Staubli VAL3: readText.dtx

public bool bBYPASS
public bool bCycle = true
public bool bCycleEnd
bool bGetSpeed = true
bool bReadEnd
bool bReadWait
public bool bResumeCycle
bool bTxtHeadOk
public bool bWriteEnd = true
frame fPrdFrame = {x=1612.648, y=43.392, z=-88.763, rx=0.062, ry=-0.933, rz=-75.763, fatherId=world[0]}
jointRx jJointRead[100]
  [0] = {j1=8.22, j2=20.1, j3=107.19, j4=-141.77, j5=44.38, j6=150.9}
  [1] = {j1=8.22, j2=20.1, j3=107.19, j4=-141.77, j5=44.38, j6=150.9}
  [2] = {j1=10.229, j2=35.494, j3=107.593, j4=-158.624, j5=56.663, j6=165.836}
  [3] = {j1=10.423, j2=28.404, j3=105.415, j4=-155.608, j5=48.169, j6=161.142}
  [4] = {j1=-54.223, j2=64.586, j3=41.499, j4=-84.729, j5=-54.881, j6=28.938}
  [5] = {j1=-45.629, j2=26.921, j3=105.631, j4=-78.314, j5=-77.561, j6=-12.796}
  [6] = {j3=109.005, j4=80.751, j5=91.42, j6=-238.352}
  [7] = {j3=63.424, j4=82.395, j5=93.028, j6=-198.425}
  [8] = {j3=109.358, j4=80.375, j5=92.272, j6=-239.01}
  [9] = {j3=62.177, j4=82.615, j5=93.831, j6=-197.649}
public jointRx jPrdHome = {j1=40.635, j2=24.616, j3=104.715, j4=-108.663, j5=68.526, j6=132.709}
mdesc mNomSpeed = {accel=16, vel=40, decel=16, tmax=80, blend=off, leave=20, reach=20}
public mdesc mSpdOfJnt[100]
  [0] = {accel=16, vel=40, decel=16, rmax=1000, tmax=200, blend=cartesian, leave=2, reach=2}
  [1] = {accel=16, vel=40, decel=16, rmax=1000, tmax=200, blend=cartesian, leave=2, reach=2}
  [2] = {accel=16, vel=40, decel=16, rmax=1000, tmax=200, blend=cartesian, leave=2, reach=2}
  [3] = {accel=16, vel=40, decel=16, rmax=1000, tmax=200, blend=cartesian, leave=2, reach=2}
  [4] = {accel=16, vel=40, decel=16, rmax=1000, tmax=200, blend=cartesian, leave=2, reach=2}
  [5] = {accel=16, vel=40, decel=16, rmax=1000, tmax=200, blend=cartesian, leave=2, reach=2}
  [6] = {accel=16, vel=40, decel=16, rmax=1000, tmax=200, blend=cartesian, leave=2, reach=2}
  [7] = {accel=16, vel=40, decel=16, rmax=1000, tmax=200, blend=cartesian, leave=2, reach=2}
  [8] = {accel=16, vel=40, decel=16, rmax=1000, tmax=200, blend=cartesian, leave=2, reach=2}
  [9] = {accel=16, vel=40, decel=16, rmax=1000, tmax=200, blend=cartesian, leave=2, reach=2}
  [10] = {accel=16, vel=40, decel=16, rmax=1000, tmax=200, blend=cartesian, leave=2, reach=2}
  [11] = {accel=16, vel=40, decel=16, rmax=1000, tmax=200, blend=cartesian, leave=2, reach=2}
  [12] = {accel=16, vel=40, decel=16, rmax=1000, tmax=200, blend=cartesian, leave=2, reach=2}
  [13] = {accel=16, vel=40, decel=16, rmax=1000, tmax=200, blend=cartesian, leave=2, reach=2}
  [14] = {accel=16, vel=40, decel=16, rmax=1000, tmax=200, blend=cartesian, leave=2, reach=2}
  [15] = {accel=16, vel=40, decel=16, rmax=1000, tmax=200, blend=cartesian, leave=2, reach=2}
  [16] = {accel=16, vel=40, decel=16, rmax=1000, tmax=200, blend=cartesian, leave=2, reach=2}
  [17] = {accel=16, vel=40, decel=16, rmax=1000, tmax=200, blend=cartesian, leave=2, reach=2}
  [18] = {accel=16, vel=40, decel=16, rmax=1000, tmax=200, blend=cartesian, leave=2, reach=2}
  [19] = {accel=16, vel=40, decel=16, rmax=1000, tmax=200, blend=cartesian, leave=2, reach=2}
  [20] = {accel=16, vel=40, decel=16, rmax=1000, tmax=200, blend=cartesian, leave=2, reach=2}
  [21] = {accel=16, vel=40, decel=16, rmax=1000, tmax=200, blend=cartesian, leave=2, reach=2}
  [22] = {accel=16, vel=40, decel=16, rmax=1000, tmax=200, blend=cartesian, leave=2, reach=2}
  [23] = {accel=16, vel=40, decel=16, rmax=1000, tmax=200, blend=cartesian, leave=2, reach=2}
  [24] = {accel=16, vel=40, decel=16, rmax=1000, tmax=200, blend=cartesian, leave=2, reach=2}
  [25] = {accel=16, vel=40, decel=16, rmax=1000, tmax=200, blend=cartesian, leave=2, reach=2}
  [26] = {accel=16, vel=40, decel=16, rmax=1000, tmax=200, blend=cartesian, leave=2, reach=2}
  [27] = {accel=16, vel=40, decel=16, rmax=1000, tmax=200, blend=cartesian, leave=2, reach=2}
  [28] = {accel=16, vel=40, decel=16, rmax=1000, tmax=200, blend=cartesian, leave=2, reach=2}
  [29] = {accel=16, vel=40, decel=16, rmax=1000, tmax=200, blend=cartesian, leave=2, reach=2}
  [30] = {accel=16, vel=40, decel=16, rmax=1000, tmax=200, blend=cartesian, leave=2, reach=2}
  [31] = {accel=16, vel=40, decel=16, rmax=1000, tmax=200, blend=cartesian, leave=2, reach=2}
  [32] = {accel=16, vel=40, decel=16, rmax=1000, tmax=200, blend=cartesian, leave=2, reach=2}
  [33] = {accel=16, vel=40, decel=16, rmax=1000, tmax=200, blend=cartesian, leave=2, reach=2}
  [34] = {accel=16, vel=40, decel=16, rmax=1000, tmax=200, blend=cartesian, leave=2, reach=2}
  [35] = {accel=16, vel=40, decel=16, rmax=1000, tmax=200, blend=cartesian, leave=2, reach=2}
  [36] = {accel=16, vel=40, decel=16, rmax=1000, tmax=200, blend=cartesian, leave=2, reach=2}
  [37] = {accel=16, vel=40, decel=16, rmax=1000, tmax=200, blend=cartesian, leave=2, reach=2}
  [38] = {accel=16, vel=40, decel=16, rmax=1000, tmax=200, blend=cartesian, leave=2, reach=2}
  [39] = {accel=16, vel=40, decel=16, rmax=1000, tmax=200, blend=cartesian, leave=2, reach=2}
  [40] = {accel=16, vel=40, decel=16, rmax=1000, tmax=200, blend=cartesian, leave=2, reach=2}
  [41] = {accel=16, vel=40, decel=16, rmax=1000, tmax=200, blend=cartesian, leave=2, reach=2}
  [42] = {accel=16, vel=40, decel=16, rmax=1000, tmax=200, blend=cartesian, leave=2, reach=2}
  [43] = {accel=16, vel=40, decel=16, rmax=1000, tmax=200, blend=cartesian, leave=2, reach=2}
  [44] = {accel=16, vel=40, decel=16, rmax=1000, tmax=200, blend=cartesian, leave=2, reach=2}
  [45] = {accel=16, vel=40, decel=16, rmax=1000, tmax=200, blend=cartesian, leave=2, reach=2}
  [46] = {accel=16, vel=40, decel=16, rmax=1000, tmax=200, blend=cartesian, leave=2, reach=2}
  [47] = {accel=16, vel=40, decel=16, rmax=1000, tmax=200, blend=cartesian, leave=2, reach=2}
  [48] = {accel=16, vel=40, decel=16, rmax=1000, tmax=200, blend=cartesian, leave=2, reach=2}
  [49] = {accel=16, vel=40, decel=16, rmax=1000, tmax=200, blend=cartesian, leave=2, reach=2}
  [50] = {accel=16, vel=40, decel=16, rmax=1000, tmax=200, blend=cartesian, leave=2, reach=2}
  [51] = {accel=16, vel=40, decel=16, rmax=1000, tmax=200, blend=cartesian, leave=2, reach=2}
  [52] = {accel=16, vel=40, decel=16, rmax=1000, tmax=200, blend=cartesian, leave=2, reach=2}
  [53] = {accel=16, vel=40, decel=16, rmax=1000, tmax=200, blend=cartesian, leave=2, reach=2}
  [54] = {accel=16, vel=40, decel=16, rmax=1000, tmax=200, blend=cartesian, leave=2, reach=2}
  [55] = {accel=16, vel=40, decel=16, rmax=1000, tmax=200, blend=cartesian, leave=2, reach=2}
  [56] = {accel=16, vel=40, decel=16, rmax=1000, tmax=200, blend=cartesian, leave=2, reach=2}
  [57] = {accel=16, vel=40, decel=16, rmax=1000, tmax=200, blend=cartesian, leave=2, reach=2}
  [58] = {accel=16, vel=40, decel=16, rmax=1000, tmax=200, blend=cartesian, leave=2, reach=2}
  [59] = {accel=16, vel=40, decel=16, rmax=1000, tmax=200, blend=cartesian, leave=2, reach=2}
  [60] = {accel=16, vel=40, decel=16, rmax=1000, tmax=200, blend=cartesian, leave=2, reach=2}
  [61] = {accel=16, vel=40, decel=16, rmax=1000, tmax=200, blend=cartesian, leave=2, reach=2}
  [62] = {accel=16, vel=40, decel=16, rmax=1000, tmax=200, blend=cartesian, leave=2, reach=2}
  [63] = {accel=16, vel=40, decel=16, rmax=1000, tmax=200, blend=cartesian, leave=2, reach=2}
  [64] = {accel=16, vel=40, decel=16, rmax=1000, tmax=200, blend=cartesian, leave=2, reach=2}
  [65] = {accel=16, vel=40, decel=16, rmax=1000, tmax=200, blend=cartesian, leave=2, reach=2}
  [66] = {accel=16, vel=40, decel=16, rmax=1000, tmax=200, blend=cartesian, leave=2, reach=2}
  [67] = {accel=16, vel=40, decel=16, rmax=1000, tmax=200, blend=cartesian, leave=2, reach=2}
  [68] = {accel=16, vel=40, decel=16, rmax=1000, tmax=200, blend=cartesian, leave=2, reach=2}
  [69] = {accel=16, vel=40, decel=16, rmax=1000, tmax=200, blend=cartesian, leave=2, reach=2}
  [70] = {accel=16, vel=40, decel=16, rmax=1000, tmax=200, blend=cartesian, leave=2, reach=2}
  [71] = {accel=16, vel=40, decel=16, rmax=1000, tmax=200, blend=cartesian, leave=2, reach=2}
  [72] = {accel=16, vel=40, decel=16, rmax=1000, tmax=200, blend=cartesian, leave=2, reach=2}
  [73] = {accel=16, vel=40, decel=16, rmax=1000, tmax=200, blend=cartesian, leave=2, reach=2}
  [74] = {accel=16, vel=40, decel=16, rmax=1000, tmax=200, blend=cartesian, leave=2, reach=2}
  [75] = {accel=16, vel=40, decel=16, rmax=1000, tmax=200, blend=cartesian, leave=2, reach=2}
  [76] = {accel=16, vel=40, decel=16, rmax=1000, tmax=200, blend=cartesian, leave=2, reach=2}
  [77] = {accel=16, vel=40, decel=16, rmax=1000, tmax=200, blend=cartesian, leave=2, reach=2}
  [78] = {accel=16, vel=40, decel=16, rmax=1000, tmax=200, blend=cartesian, leave=2, reach=2}
  [79] = {accel=16, vel=40, decel=16, rmax=1000, tmax=200, blend=cartesian, leave=2, reach=2}
  [80] = {accel=16, vel=40, decel=16, rmax=1000, tmax=200, blend=cartesian, leave=2, reach=2}
  [81] = {accel=16, vel=40, decel=16, rmax=1000, tmax=200, blend=cartesian, leave=2, reach=2}
  [82] = {accel=16, vel=40, decel=16, rmax=1000, tmax=200, blend=cartesian, leave=2, reach=2}
  [83] = {accel=16, vel=40, decel=16, rmax=1000, tmax=200, blend=cartesian, leave=2, reach=2}
  [84] = {accel=16, vel=40, decel=16, rmax=1000, tmax=200, blend=cartesian, leave=2, reach=2}
  [85] = {accel=16, vel=40, decel=16, rmax=1000, tmax=200, blend=cartesian, leave=2, reach=2}
  [86] = {accel=16, vel=40, decel=16, rmax=1000, tmax=200, blend=cartesian, leave=2, reach=2}
  [87] = {accel=16, vel=40, decel=16, rmax=1000, tmax=200, blend=cartesian, leave=2, reach=2}
  [88] = {accel=16, vel=40, decel=16, rmax=1000, tmax=200, blend=cartesian, leave=2, reach=2}
  [89] = {accel=16, vel=40, decel=16, rmax=1000, tmax=200, blend=cartesian, leave=2, reach=2}
  [90] = {accel=16, vel=40, decel=16, rmax=1000, tmax=200, blend=cartesian, leave=2, reach=2}
  [91] = {accel=16, vel=40, decel=16, rmax=1000, tmax=200, blend=cartesian, leave=2, reach=2}
  [92] = {accel=16, vel=40, decel=16, rmax=1000, tmax=200, blend=cartesian, leave=2, reach=2}
  [93] = {accel=16, vel=40, decel=16, rmax=1000, tmax=200, blend=cartesian, leave=2, reach=2}
  [94] = {accel=16, vel=40, decel=16, rmax=1000, tmax=200, blend=cartesian, leave=2, reach=2}
  [95] = {accel=16, vel=40, decel=16, rmax=1000, tmax=200, blend=cartesian, leave=2, reach=2}
  [96] = {accel=16, vel=40, decel=16, rmax=1000, tmax=200, blend=cartesian, leave=2, reach=2}
  [97] = {accel=16, vel=40, decel=16, rmax=1000, tmax=200, blend=cartesian, leave=2, reach=2}
  [98] = {accel=16, vel=40, decel=16, rmax=1000, tmax=200, blend=cartesian, leave=2, reach=2}
  [99] = {accel=16, vel=40, decel=16, rmax=1000, tmax=200, blend=cartesian, leave=2, reach=2}
public mdesc mSpdOfPt[1000]
  [0] = {accel=40, decel=4000, tmax=15.672, leave=0, reach=0.5}
  [1] = {accel=40, decel=4000, tmax=16.369, leave=0, reach=0.5}
  [2] = {accel=40, decel=4000, tmax=17.023, leave=0, reach=0.5}
  [3] = {accel=40, decel=4000, tmax=17.611, leave=0, reach=0.5}
  [4] = {accel=40, decel=4000, tmax=18.123, leave=0, reach=0.5}
  [5] = {accel=40, decel=4000, tmax=18.562, leave=0, reach=0.5}
  [6] = {accel=40, decel=4000, tmax=18.942, leave=0, reach=0.5}
  [7] = {accel=40, decel=4000, tmax=19.269, leave=0, reach=0.5}
  [8] = {accel=40, decel=4000, tmax=19.551, leave=0, reach=0.5}
  [9] = {accel=40, decel=4000, tmax=19.789, leave=0, reach=0.5}
  [10] = {accel=40, decel=4000, tmax=19.988, leave=0, reach=0.5}
  [11] = {accel=40, decel=4000, tmax=20.148, leave=0, reach=0.5}
  [12] = {accel=40, decel=4000, tmax=20.275, leave=0, reach=0.5}
  [13] = {accel=40, decel=4000, tmax=20.376, leave=0, reach=0.5}
  [14] = {accel=40, decel=4000, tmax=20.455, leave=0, reach=0.5}
  [15] = {accel=40, decel=4000, tmax=20.517, leave=0, reach=0.5}
  [16] = {accel=40, decel=4000, tmax=20.563, leave=0, reach=0.5}
  [17] = {accel=40, decel=4000, tmax=20.596, leave=0, reach=0.5}
  [18] = {accel=40, decel=4000, tmax=20.615, leave=0, reach=0.5}
  [19] = {accel=40, decel=4000, tmax=20.621, leave=0, reach=0.5}
  [20] = {accel=40, decel=4000, tmax=20.615, leave=0, reach=0.5}
  [21] = {accel=40, decel=4000, tmax=20.6, leave=0, reach=0.5}
  [22] = {accel=40, decel=4000, tmax=20.583, leave=0, reach=0.5}
  [23] = {accel=40, decel=4000, tmax=20.564, leave=0, reach=0.5}
  [24] = {accel=40, decel=4000, tmax=20.543, leave=0, reach=0.5}
  [25] = {accel=40, decel=4000, tmax=20.52, leave=0, reach=0.5}
  [26] = {accel=40, decel=4000, tmax=20.501, leave=0, reach=0.5}
  [27] = {accel=40, decel=4000, tmax=20.495, leave=0, reach=0.5}
  [28] = {accel=40, decel=4000, tmax=20.506, leave=0, reach=0.5}
  [29] = {accel=40, decel=4000, tmax=20.53, leave=0, reach=0.5}
  [30] = {accel=40, decel=4000, tmax=20.554, leave=0, reach=0.5}
  [31] = {accel=40, decel=4000, tmax=20.568, leave=0, reach=0.5}
  [32] = {accel=40, decel=4000, tmax=20.569, leave=0, reach=0.5}
  [33] = {accel=40, decel=4000, tmax=20.562, leave=0, reach=0.5}
  [34] = {accel=40, decel=4000, tmax=20.56, leave=0, reach=0.5}
  [35] = {accel=40, decel=4000, tmax=20.571, leave=0, reach=0.5}
  [36] = {accel=40, decel=4000, tmax=20.59, leave=0, reach=0.5}
  [37] = {accel=40, decel=4000, tmax=20.611, leave=0, reach=0.5}
  [38] = {accel=40, decel=4000, tmax=20.641, leave=0, reach=0.5}
  [39] = {accel=40, decel=4000, tmax=20.701, leave=0, reach=0.5}
  [40] = {accel=40, decel=4000, tmax=20.817, leave=0, reach=0.5}
  [41] = {accel=40, decel=4000, tmax=20.998, leave=0, reach=0.5}
  [42] = {accel=40, decel=4000, tmax=21.232, leave=0, reach=0.5}
  [43] = {accel=40, decel=4000, tmax=21.485, leave=0, reach=0.5}
  [44] = {accel=40, decel=4000, tmax=21.717, leave=0, reach=0.5}
  [45] = {accel=40, decel=4000, tmax=21.897, leave=0, reach=0.5}
  [46] = {accel=40, decel=4000, tmax=22.019, leave=0, reach=0.5}
  [47] = {accel=40, decel=4000, tmax=22.098, leave=0, reach=0.5}
  [48] = {accel=40, decel=4000, tmax=22.154, leave=0, reach=0.5}
  [49] = {accel=40, decel=4000, tmax=22.195, leave=0, reach=0.5}
  [50] = {accel=40, decel=4000, tmax=22.217, leave=0, reach=0.5}
  [51] = {accel=40, decel=4000, tmax=22.213, leave=0, reach=0.5}
  [52] = {accel=40, decel=4000, tmax=22.189, leave=0, reach=0.5}
  [53] = {accel=40, decel=4000, tmax=22.153, leave=0, reach=0.5}
  [54] = {accel=40, decel=4000, tmax=22.116, leave=0, reach=0.5}
  [55] = {accel=40, decel=4000, tmax=22.079, leave=0, reach=0.5}
  [56] = {accel=40, decel=4000, tmax=22.04, leave=0, reach=0.5}
  [57] = {accel=40, decel=4000, tmax=21.995, leave=0, reach=0.5}
  [58] = {accel=40, decel=4000, tmax=21.94, leave=0, reach=0.5}
  [59] = {accel=40, decel=4000, tmax=21.876, leave=0, reach=0.5}
  [60] = {accel=40, decel=4000, tmax=21.809, leave=0, reach=0.5}
  [61] = {accel=40, decel=4000, tmax=21.74, leave=0, reach=0.5}
  [62] = {accel=40, decel=4000, tmax=21.667, leave=0, reach=0.5}
  [63] = {accel=40, decel=4000, tmax=21.585, leave=0, reach=0.5}
  [64] = {accel=40, decel=4000, tmax=21.491, leave=0, reach=0.5}
  [65] = {accel=40, decel=4000, tmax=21.382, leave=0, reach=0.5}
  [66] = {accel=40, decel=4000, tmax=21.258, leave=0, reach=0.5}
  [67] = {accel=40, decel=4000, tmax=21.117, leave=0, reach=0.5}
  [68] = {accel=40, decel=4000, tmax=20.955, leave=0, reach=0.5}
  [69] = {accel=40, decel=4000, tmax=20.766, leave=0, reach=0.5}
  [70] = {accel=40, decel=4000, tmax=20.55, leave=0, reach=0.5}
  [71] = {accel=40, decel=4000, tmax=20.313, leave=0, reach=0.5}
  [72] = {accel=40, decel=4000, tmax=20.06, leave=0, reach=0.5}
  [73] = {accel=40, decel=4000, tmax=19.795, leave=0, reach=0.5}
  [74] = {accel=40, decel=4000, tmax=19.518, leave=0, reach=0.5}
  [75] = {accel=40, decel=4000, tmax=19.229, leave=0, reach=0.5}
  [76] = {accel=40, decel=4000, tmax=18.929, leave=0, reach=0.5}
  [77] = {accel=40, decel=4000, tmax=18.616, leave=0, reach=0.5}
  [78] = {accel=40, decel=4000, tmax=18.288, leave=0, reach=0.5}
  [79] = {accel=40, decel=4000, tmax=17.947, leave=0, reach=0.5}
  [80] = {accel=40, decel=4000, tmax=17.601, leave=0, reach=0.5}
  [81] = {accel=40, decel=4000, tmax=17.259, leave=0, reach=0.5}
  [82] = {accel=40, decel=4000, tmax=16.931, leave=0, reach=0.5}
  [83] = {accel=40, decel=4000, tmax=16.613, leave=0, reach=0.5}
  [84] = {accel=40, decel=4000, tmax=16.293, leave=0, reach=0.5}
  [85] = {accel=40, decel=4000, tmax=15.957, leave=0, reach=0.5}
  [86] = {accel=40, decel=4000, tmax=15.595, leave=0, reach=0.5}
  [87] = {accel=40, decel=4000, tmax=15.202, leave=0, reach=0.5}
  [88] = {accel=40, decel=4000, tmax=14.779, leave=0, reach=0.5}
  [89] = {accel=40, decel=4000, tmax=14.331, leave=0, reach=0.5}
  [90] = {accel=40, decel=4000, tmax=13.865, leave=0, reach=0.5}
  [91] = {accel=40, decel=4000, tmax=13.393, leave=0, reach=0.5}
  [92] = {accel=40, decel=4000, tmax=12.925, leave=0, reach=0.5}
  [93] = {accel=40, decel=4000, tmax=28.624, leave=0, reach=0.5}
  [94] = {accel=40, decel=4000, tmax=13.153, leave=0, reach=0.5}
  [95] = {accel=40, decel=4000, tmax=13.601, leave=0, reach=0.5}
  [96] = {accel=40, decel=4000, tmax=14.047, leave=0, reach=0.5}
  [97] = {accel=40, decel=4000, tmax=14.484, leave=0, reach=0.5}
  [98] = {accel=40, decel=4000, tmax=14.903, leave=0, reach=0.5}
  [99] = {accel=40, decel=4000, tmax=15.299, leave=0, reach=0.5}
  [100] = {accel=40, decel=4000, tmax=15.67, leave=0, reach=0.5}
  [101] = {accel=40, decel=4000, tmax=16.022, leave=0, reach=0.5}
  [102] = {accel=40, decel=4000, tmax=16.368, leave=0, reach=0.5}
  [103] = {accel=40, decel=4000, tmax=16.723, leave=0, reach=0.5}
  [104] = {accel=40, decel=4000, tmax=17.091, leave=0, reach=0.5}
  [105] = {accel=40, decel=4000, tmax=17.467, leave=0, reach=0.5}
  [106] = {accel=40, decel=4000, tmax=17.843, leave=0, reach=0.5}
  [107] = {accel=40, decel=4000, tmax=18.211, leave=0, reach=0.5}
  [108] = {accel=40, decel=4000, tmax=18.567, leave=0, reach=0.5}
  [109] = {accel=40, decel=4000, tmax=18.911, leave=0, reach=0.5}
  [110] = {accel=40, decel=4000, tmax=19.238, leave=0, reach=0.5}
  [111] = {accel=40, decel=4000, tmax=19.547, leave=0, reach=0.5}
  [112] = {accel=40, decel=4000, tmax=19.837, leave=0, reach=0.5}
  [113] = {accel=40, decel=4000, tmax=20.111, leave=0, reach=0.5}
  [114] = {accel=40, decel=4000, tmax=20.367, leave=0, reach=0.5}
  [115] = {accel=40, decel=4000, tmax=20.602, leave=0, reach=0.5}
  [116] = {accel=40, decel=4000, tmax=20.813, leave=0, reach=0.5}
  [117] = {accel=40, decel=4000, tmax=21.001, leave=0, reach=0.5}
  [118] = {accel=40, decel=4000, tmax=21.172, leave=0, reach=0.5}
  [119] = {accel=40, decel=4000, tmax=21.328, leave=0, reach=0.5}
  [120] = {accel=40, decel=4000, tmax=21.469, leave=0, reach=0.5}
  [121] = {accel=40, decel=4000, tmax=21.595, leave=0, reach=0.5}
  [122] = {accel=40, decel=4000, tmax=21.708, leave=0, reach=0.5}
  [123] = {accel=40, decel=4000, tmax=21.81, leave=0, reach=0.5}
  [124] = {accel=40, decel=4000, tmax=21.907, leave=0, reach=0.5}
  [125] = {accel=40, decel=4000, tmax=21.998, leave=0, reach=0.5}
  [126] = {accel=40, decel=4000, tmax=22.082, leave=0, reach=0.5}
  [127] = {accel=40, decel=4000, tmax=22.155, leave=0, reach=0.5}
  [128] = {accel=40, decel=4000, tmax=22.217, leave=0, reach=0.5}
  [129] = {accel=40, decel=4000, tmax=22.272, leave=0, reach=0.5}
  [130] = {accel=40, decel=4000, tmax=22.324, leave=0, reach=0.5}
  [131] = {accel=40, decel=4000, tmax=22.375, leave=0, reach=0.5}
  [132] = {accel=40, decel=4000, tmax=22.423, leave=0, reach=0.5}
  [133] = {accel=40, decel=4000, tmax=22.459, leave=0, reach=0.5}
  [134] = {accel=40, decel=4000, tmax=22.473, leave=0, reach=0.5}
  [135] = {accel=40, decel=4000, tmax=22.461, leave=0, reach=0.5}
  [136] = {accel=40, decel=4000, tmax=22.43, leave=0, reach=0.5}
  [137] = {accel=40, decel=4000, tmax=22.386, leave=0, reach=0.5}
  [138] = {accel=40, decel=4000, tmax=22.324, leave=0, reach=0.5}
  [139] = {accel=40, decel=4000, tmax=22.223, leave=0, reach=0.5}
  [140] = {accel=40, decel=4000, tmax=22.065, leave=0, reach=0.5}
  [141] = {accel=40, decel=4000, tmax=21.849, leave=0, reach=0.5}
  [142] = {accel=40, decel=4000, tmax=21.606, leave=0, reach=0.5}
  [143] = {accel=40, decel=4000, tmax=21.378, leave=0, reach=0.5}
  [144] = {accel=40, decel=4000, tmax=21.204, leave=0, reach=0.5}
  [145] = {accel=40, decel=4000, tmax=21.097, leave=0, reach=0.5}
  [146] = {accel=40, decel=4000, tmax=21.048, leave=0, reach=0.5}
  [147] = {accel=40, decel=4000, tmax=21.033, leave=0, reach=0.5}
  [148] = {accel=40, decel=4000, tmax=21.031, leave=0, reach=0.5}
  [149] = {accel=40, decel=4000, tmax=21.033, leave=0, reach=0.5}
  [150] = {accel=40, decel=4000, tmax=21.04, leave=0, reach=0.5}
  [151] = {accel=40, decel=4000, tmax=21.05, leave=0, reach=0.5}
  [152] = {accel=40, decel=4000, tmax=21.061, leave=0, reach=0.5}
  [153] = {accel=40, decel=4000, tmax=21.064, leave=0, reach=0.5}
  [154] = {accel=40, decel=4000, tmax=21.054, leave=0, reach=0.5}
  [155] = {accel=40, decel=4000, tmax=21.033, leave=0, reach=0.5}
  [156] = {accel=40, decel=4000, tmax=21.011, leave=0, reach=0.5}
  [157] = {accel=40, decel=4000, tmax=20.997, leave=0, reach=0.5}
  [158] = {accel=40, decel=4000, tmax=20.992, leave=0, reach=0.5}
  [159] = {accel=40, decel=4000, tmax=20.987, leave=0, reach=0.5}
  [160] = {accel=40, decel=4000, tmax=20.974, leave=0, reach=0.5}
  [161] = {accel=40, decel=4000, tmax=20.952, leave=0, reach=0.5}
  [162] = {accel=40, decel=4000, tmax=20.927, leave=0, reach=0.5}
  [163] = {accel=40, decel=4000, tmax=20.9, leave=0, reach=0.5}
  [164] = {accel=40, decel=4000, tmax=20.867, leave=0, reach=0.5}
  [165] = {accel=40, decel=4000, tmax=20.817, leave=0, reach=0.5}
  [166] = {accel=40, decel=4000, tmax=20.744, leave=0, reach=0.5}
  [167] = {accel=40, decel=4000, tmax=20.65, leave=0, reach=0.5}
  [168] = {accel=40, decel=4000, tmax=20.537, leave=0, reach=0.5}
  [169] = {accel=40, decel=4000, tmax=20.405, leave=0, reach=0.5}
  [170] = {accel=40, decel=4000, tmax=20.254, leave=0, reach=0.5}
  [171] = {accel=40, decel=4000, tmax=20.081, leave=0, reach=0.5}
  [172] = {accel=40, decel=4000, tmax=19.882, leave=0, reach=0.5}
  [173] = {accel=40, decel=4000, tmax=19.655, leave=0, reach=0.5}
  [174] = {accel=40, decel=4000, tmax=19.393, leave=0, reach=0.5}
  [175] = {accel=40, decel=4000, tmax=19.098, leave=0, reach=0.5}
  [176] = {accel=40, decel=4000, tmax=18.769, leave=0, reach=0.5}
  [177] = {accel=40, decel=4000, tmax=18.404, leave=0, reach=0.5}
  [178] = {accel=40, decel=4000, tmax=17.999, leave=0, reach=0.5}
  [179] = {accel=40, decel=4000, tmax=17.549, leave=0, reach=0.5}
  [180] = {accel=40, decel=4000, tmax=17.05, leave=0, reach=0.5}
  [181] = {accel=40, decel=4000, tmax=16.497, leave=0, reach=0.5}
  [182] = {accel=40, decel=4000, tmax=15.886, leave=0, reach=0.5}
  [183] = {accel=40, decel=4000, tmax=34.921, leave=0, reach=0.5}
  [184] = {accel=40, decel=4000, tmax=15.966, leave=0, reach=0.5}
  [185] = {accel=40, decel=4000, tmax=16.507, leave=0, reach=0.5}
  [186] = {accel=40, decel=4000, tmax=17.012, leave=0, reach=0.5}
  [187] = {accel=40, decel=4000, tmax=17.481, leave=0, reach=0.5}
  [188] = {accel=40, decel=4000, tmax=17.915, leave=0, reach=0.5}
  [189] = {accel=40, decel=4000, tmax=18.317, leave=0, reach=0.5}
  [190] = {accel=40, decel=4000, tmax=18.687, leave=0, reach=0.5}
  [191] = {accel=40, decel=4000, tmax=19.026, leave=0, reach=0.5}
  [192] = {accel=40, decel=4000, tmax=19.333, leave=0, reach=0.5}
  [193] = {accel=40, decel=4000, tmax=19.612, leave=0, reach=0.5}
  [194] = {accel=40, decel=4000, tmax=19.868, leave=0, reach=0.5}
  [195] = {accel=40, decel=4000, tmax=20.105, leave=0, reach=0.5}
  [196] = {accel=40, decel=4000, tmax=20.322, leave=0, reach=0.5}
  [197] = {accel=40, decel=4000, tmax=20.52, leave=0, reach=0.5}
  [198] = {accel=40, decel=4000, tmax=20.694, leave=0, reach=0.5}
  [199] = {accel=40, decel=4000, tmax=20.835, leave=0, reach=0.5}
  [200] = {accel=40, decel=4000, tmax=20.941, leave=0, reach=0.5}
  [201] = {accel=40, decel=4000, tmax=21.018, leave=0, reach=0.5}
  [202] = {accel=40, decel=4000, tmax=21.084, leave=0, reach=0.5}
  [203] = {accel=40, decel=4000, tmax=21.153, leave=0, reach=0.5}
  [204] = {accel=40, decel=4000, tmax=21.221, leave=0, reach=0.5}
  [205] = {accel=40, decel=4000, tmax=21.279, leave=0, reach=0.5}
  [206] = {accel=40, decel=4000, tmax=21.32, leave=0, reach=0.5}
  [207] = {accel=40, decel=4000, tmax=21.347, leave=0, reach=0.5}
  [208] = {accel=40, decel=4000, tmax=21.367, leave=0, reach=0.5}
  [209] = {accel=40, decel=4000, tmax=21.386, leave=0, reach=0.5}
  [210] = {accel=40, decel=4000, tmax=21.4, leave=0, reach=0.5}
  [211] = {accel=40, decel=4000, tmax=21.406, leave=0, reach=0.5}
  [212] = {accel=40, decel=4000, tmax=21.403, leave=0, reach=0.5}
  [213] = {accel=40, decel=4000, tmax=21.393, leave=0, reach=0.5}
  [214] = {accel=40, decel=4000, tmax=21.381, leave=0, reach=0.5}
  [215] = {accel=40, decel=4000, tmax=21.369, leave=0, reach=0.5}
  [216] = {accel=40, decel=4000, tmax=21.359, leave=0, reach=0.5}
  [217] = {accel=40, decel=4000, tmax=21.354, leave=0, reach=0.5}
  [218] = {accel=40, decel=4000, tmax=21.364, leave=0, reach=0.5}
  [219] = {accel=40, decel=4000, tmax=21.408, leave=0, reach=0.5}
  [220] = {accel=40, decel=4000, tmax=21.506, leave=0, reach=0.5}
  [221] = {accel=40, decel=4000, tmax=21.663, leave=0, reach=0.5}
  [222] = {accel=40, decel=4000, tmax=21.866, leave=0, reach=0.5}
  [223] = {accel=40, decel=4000, tmax=22.075, leave=0, reach=0.5}
  [224] = {accel=40, decel=4000, tmax=22.25, leave=0, reach=0.5}
  [225] = {accel=40, decel=4000, tmax=22.368, leave=0, reach=0.5}
  [226] = {accel=40, decel=4000, tmax=22.439, leave=0, reach=0.5}
  [227] = {accel=40, decel=4000, tmax=22.485, leave=0, reach=0.5}
  [228] = {accel=40, decel=4000, tmax=22.523, leave=0, reach=0.5}
  [229] = {accel=40, decel=4000, tmax=22.553, leave=0, reach=0.5}
  [230] = {accel=40, decel=4000, tmax=22.566, leave=0, reach=0.5}
  [231] = {accel=40, decel=4000, tmax=22.552, leave=0, reach=0.5}
  [232] = {accel=40, decel=4000, tmax=22.512, leave=0, reach=0.5}
  [233] = {accel=40, decel=4000, tmax=22.455, leave=0, reach=0.5}
  [234] = {accel=40, decel=4000, tmax=22.392, leave=0, reach=0.5}
  [235] = {accel=40, decel=4000, tmax=22.327, leave=0, reach=0.5}
  [236] = {accel=40, decel=4000, tmax=22.257, leave=0, reach=0.5}
  [237] = {accel=40, decel=4000, tmax=22.178, leave=0, reach=0.5}
  [238] = {accel=40, decel=4000, tmax=22.085, leave=0, reach=0.5}
  [239] = {accel=40, decel=4000, tmax=21.979, leave=0, reach=0.5}
  [240] = {accel=40, decel=4000, tmax=21.864, leave=0, reach=0.5}
  [241] = {accel=40, decel=4000, tmax=21.743, leave=0, reach=0.5}
  [242] = {accel=40, decel=4000, tmax=21.613, leave=0, reach=0.5}
  [243] = {accel=40, decel=4000, tmax=21.472, leave=0, reach=0.5}
  [244] = {accel=40, decel=4000, tmax=21.316, leave=0, reach=0.5}
  [245] = {accel=40, decel=4000, tmax=21.144, leave=0, reach=0.5}
  [246] = {accel=40, decel=4000, tmax=20.958, leave=0, reach=0.5}
  [247] = {accel=40, decel=4000, tmax=20.76, leave=0, reach=0.5}
  [248] = {accel=40, decel=4000, tmax=20.548, leave=0, reach=0.5}
  [249] = {accel=40, decel=4000, tmax=20.318, leave=0, reach=0.5}
  [250] = {accel=40, decel=4000, tmax=20.069, leave=0, reach=0.5}
  [251] = {accel=40, decel=4000, tmax=19.799, leave=0, reach=0.5}
  [252] = {accel=40, decel=4000, tmax=19.511, leave=0, reach=0.5}
  [253] = {accel=40, decel=4000, tmax=19.202, leave=0, reach=0.5}
  [254] = {accel=40, decel=4000, tmax=18.868, leave=0, reach=0.5}
  [255] = {accel=40, decel=4000, tmax=18.508, leave=0, reach=0.5}
  [256] = {accel=40, decel=4000, tmax=18.128, leave=0, reach=0.5}
  [257] = {accel=40, decel=4000, tmax=17.735, leave=0, reach=0.5}
  [258] = {accel=40, decel=4000, tmax=17.333, leave=0, reach=0.5}
  [259] = {accel=40, decel=4000, tmax=16.925, leave=0, reach=0.5}
  [260] = {accel=40, decel=4000, tmax=16.52, leave=0, reach=0.5}
  [261] = {accel=40, decel=4000, tmax=16.124, leave=0, reach=0.5}
  [262] = {accel=40, decel=4000, tmax=15.739, leave=0, reach=0.5}
  [263] = {accel=40, decel=4000, tmax=15.36, leave=0, reach=0.5}
  [264] = {accel=40, decel=4000, tmax=14.977, leave=0, reach=0.5}
  [265] = {accel=40, decel=4000, tmax=14.58, leave=0, reach=0.5}
  [266] = {accel=40, decel=4000, tmax=14.169, leave=0, reach=0.5}
  [267] = {accel=40, decel=4000, tmax=13.749, leave=0, reach=0.5}
  [268] = {accel=40, decel=4000, tmax=13.325, leave=0, reach=0.5}
  [269] = {accel=40, decel=4000, tmax=29.431, leave=0, reach=0.5}
  [270] = {accel=40, decel=4000, tmax=13.43, leave=0, reach=0.5}
  [271] = {accel=40, decel=4000, tmax=13.831, leave=0, reach=0.5}
  [272] = {accel=40, decel=4000, tmax=14.232, leave=0, reach=0.5}
  [273] = {accel=40, decel=4000, tmax=14.633, leave=0, reach=0.5}
  [274] = {accel=40, decel=4000, tmax=15.039, leave=0, reach=0.5}
  [275] = {accel=40, decel=4000, tmax=15.454, leave=0, reach=0.5}
  [276] = {accel=40, decel=4000, tmax=15.879, leave=0, reach=0.5}
  [277] = {accel=40, decel=4000, tmax=16.311, leave=0, reach=0.5}
  [278] = {accel=40, decel=4000, tmax=16.744, leave=0, reach=0.5}
  [279] = {accel=40, decel=4000, tmax=17.173, leave=0, reach=0.5}
  [280] = {accel=40, decel=4000, tmax=17.594, leave=0, reach=0.5}
  [281] = {accel=40, decel=4000, tmax=18.002, leave=0, reach=0.5}
  [282] = {accel=40, decel=4000, tmax=18.387, leave=0, reach=0.5}
  [283] = {accel=40, decel=4000, tmax=18.742, leave=0, reach=0.5}
  [284] = {accel=40, decel=4000, tmax=19.067, leave=0, reach=0.5}
  [285] = {accel=40, decel=4000, tmax=19.367, leave=0, reach=0.5}
  [286] = {accel=40, decel=4000, tmax=19.646, leave=0, reach=0.5}
  [287] = {accel=40, decel=4000, tmax=19.908, leave=0, reach=0.5}
  [288] = {accel=40, decel=4000, tmax=20.154, leave=0, reach=0.5}
  [289] = {accel=40, decel=4000, tmax=20.386, leave=0, reach=0.5}
  [290] = {accel=40, decel=4000, tmax=20.608, leave=0, reach=0.5}
  [291] = {accel=40, decel=4000, tmax=20.821, leave=0, reach=0.5}
  [292] = {accel=40, decel=4000, tmax=21.021, leave=0, reach=0.5}
  [293] = {accel=40, decel=4000, tmax=21.206, leave=0, reach=0.5}
  [294] = {accel=40, decel=4000, tmax=21.373, leave=0, reach=0.5}
  [295] = {accel=40, decel=4000, tmax=21.528, leave=0, reach=0.5}
  [296] = {accel=40, decel=4000, tmax=21.673, leave=0, reach=0.5}
  [297] = {accel=40, decel=4000, tmax=21.809, leave=0, reach=0.5}
  [298] = {accel=40, decel=4000, tmax=21.934, leave=0, reach=0.5}
  [299] = {accel=40, decel=4000, tmax=22.042, leave=0, reach=0.5}
  [300] = {accel=40, decel=4000, tmax=22.134, leave=0, reach=0.5}
  [301] = {accel=40, decel=4000, tmax=22.213, leave=0, reach=0.5}
  [302] = {accel=40, decel=4000, tmax=22.287, leave=0, reach=0.5}
  [303] = {accel=40, decel=4000, tmax=22.358, leave=0, reach=0.5}
  [304] = {accel=40, decel=4000, tmax=22.421, leave=0, reach=0.5}
  [305] = {accel=40, decel=4000, tmax=22.463, leave=0, reach=0.5}
  [306] = {accel=40, decel=4000, tmax=22.473, leave=0, reach=0.5}
  [307] = {accel=40, decel=4000, tmax=22.453, leave=0, reach=0.5}
  [308] = {accel=40, decel=4000, tmax=22.416, leave=0, reach=0.5}
  [309] = {accel=40, decel=4000, tmax=22.378, leave=0, reach=0.5}
  [310] = {accel=40, decel=4000, tmax=22.342, leave=0, reach=0.5}
  [311] = {accel=40, decel=4000, tmax=22.301, leave=0, reach=0.5}
  [312] = {accel=40, decel=4000, tmax=22.231, leave=0, reach=0.5}
  [313] = {accel=40, decel=4000, tmax=22.114, leave=0, reach=0.5}
  [314] = {accel=40, decel=4000, tmax=21.958, leave=0, reach=0.5}
  [315] = {accel=40, decel=4000, tmax=21.796, leave=0, reach=0.5}
  [316] = {accel=40, decel=4000, tmax=21.663, leave=0, reach=0.5}
  [317] = {accel=40, decel=4000, tmax=21.576, leave=0, reach=0.5}
  [318] = {accel=40, decel=4000, tmax=21.535, leave=0, reach=0.5}
  [319] = {accel=40, decel=4000, tmax=21.524, leave=0, reach=0.5}
  [320] = {accel=40, decel=4000, tmax=21.53, leave=0, reach=0.5}
  [321] = {accel=40, decel=4000, tmax=21.54, leave=0, reach=0.5}
  [322] = {accel=40, decel=4000, tmax=21.551, leave=0, reach=0.5}
  [323] = {accel=40, decel=4000, tmax=21.561, leave=0, reach=0.5}
  [324] = {accel=40, decel=4000, tmax=21.567, leave=0, reach=0.5}
  [325] = {accel=40, decel=4000, tmax=21.569, leave=0, reach=0.5}
  [326] = {accel=40, decel=4000, tmax=21.566, leave=0, reach=0.5}
  [327] = {accel=40, decel=4000, tmax=21.557, leave=0, reach=0.5}
  [328] = {accel=40, decel=4000, tmax=21.538, leave=0, reach=0.5}
  [329] = {accel=40, decel=4000, tmax=21.504, leave=0, reach=0.5}
  [330] = {accel=40, decel=4000, tmax=21.447, leave=0, reach=0.5}
  [331] = {accel=40, decel=4000, tmax=21.364, leave=0, reach=0.5}
  [332] = {accel=40, decel=4000, tmax=21.26, leave=0, reach=0.5}
  [333] = {accel=40, decel=4000, tmax=21.149, leave=0, reach=0.5}
  [334] = {accel=40, decel=4000, tmax=21.04, leave=0, reach=0.5}
  [335] = {accel=40, decel=4000, tmax=20.932, leave=0, reach=0.5}
  [336] = {accel=40, decel=4000, tmax=20.805, leave=0, reach=0.5}
  [337] = {accel=40, decel=4000, tmax=20.639, leave=0, reach=0.5}
  [338] = {accel=40, decel=4000, tmax=20.426, leave=0, reach=0.5}
  [339] = {accel=40, decel=4000, tmax=20.175, leave=0, reach=0.5}
  [340] = {accel=40, decel=4000, tmax=19.897, leave=0, reach=0.5}
  [341] = {accel=40, decel=4000, tmax=19.603, leave=0, reach=0.5}
  [342] = {accel=40, decel=4000, tmax=19.296, leave=0, reach=0.5}
  [343] = {accel=40, decel=4000, tmax=18.975, leave=0, reach=0.5}
  [344] = {accel=40, decel=4000, tmax=18.635, leave=0, reach=0.5}
  [345] = {accel=40, decel=4000, tmax=18.27, leave=0, reach=0.5}
  [346] = {accel=40, decel=4000, tmax=17.874, leave=0, reach=0.5}
  [347] = {accel=40, decel=4000, tmax=17.448, leave=0, reach=0.5}
  [348] = {accel=40, decel=4000, tmax=16.994, leave=0, reach=0.5}
  [349] = {accel=40, decel=4000, tmax=16.511, leave=0, reach=0.5}
  [350] = {accel=40, decel=4000, tmax=16.001, leave=0, reach=0.5}
  [351] = {accel=40, decel=4000, tmax=35.192, leave=0, reach=0.5}
  [352] = {accel=40, decel=4000, tmax=16.003, leave=0, reach=0.5}
  [353] = {accel=40, decel=4000, tmax=16.487, leave=0, reach=0.5}
  [354] = {accel=40, decel=4000, tmax=16.949, leave=0, reach=0.5}
  [355] = {accel=40, decel=4000, tmax=17.385, leave=0, reach=0.5}
  [356] = {accel=40, decel=4000, tmax=17.795, leave=0, reach=0.5}
  [357] = {accel=40, decel=4000, tmax=18.183, leave=0, reach=0.5}
  [358] = {accel=40, decel=4000, tmax=18.556, leave=0, reach=0.5}
  [359] = {accel=40, decel=4000, tmax=18.916, leave=0, reach=0.5}
  [360] = {accel=40, decel=4000, tmax=19.267, leave=0, reach=0.5}
  [361] = {accel=40, decel=4000, tmax=19.605, leave=0, reach=0.5}
  [362] = {accel=40, decel=4000, tmax=19.919, leave=0, reach=0.5}
  [363] = {accel=40, decel=4000, tmax=20.195, leave=0, reach=0.5}
  [364] = {accel=40, decel=4000, tmax=20.425, leave=0, reach=0.5}
  [365] = {accel=40, decel=4000, tmax=20.612, leave=0, reach=0.5}
  [366] = {accel=40, decel=4000, tmax=20.777, leave=0, reach=0.5}
  [367] = {accel=40, decel=4000, tmax=20.934, leave=0, reach=0.5}
  [368] = {accel=40, decel=4000, tmax=21.089, leave=0, reach=0.5}
  [369] = {accel=40, decel=4000, tmax=21.234, leave=0, reach=0.5}
  [370] = {accel=40, decel=4000, tmax=21.357, leave=0, reach=0.5}
  [371] = {accel=40, decel=4000, tmax=21.445, leave=0, reach=0.5}
  [372] = {accel=40, decel=4000, tmax=21.497, leave=0, reach=0.5}
  [373] = {accel=40, decel=4000, tmax=21.52, leave=0, reach=0.5}
  [374] = {accel=40, decel=4000, tmax=21.525, leave=0, reach=0.5}
  [375] = {accel=40, decel=4000, tmax=21.523, leave=0, reach=0.5}
  [376] = {accel=40, decel=4000, tmax=21.521, leave=0, reach=0.5}
  [377] = {accel=40, decel=4000, tmax=21.519, leave=0, reach=0.5}
  [378] = {accel=40, decel=4000, tmax=21.513, leave=0, reach=0.5}
  [379] = {accel=40, decel=4000, tmax=21.504, leave=0, reach=0.5}
  [380] = {accel=40, decel=4000, tmax=21.493, leave=0, reach=0.5}
  [381] = {accel=40, decel=4000, tmax=21.485, leave=0, reach=0.5}
  [382] = {accel=40, decel=4000, tmax=21.491, leave=0, reach=0.5}
  [383] = {accel=40, decel=4000, tmax=21.525, leave=0, reach=0.5}
  [384] = {accel=40, decel=4000, tmax=21.596, leave=0, reach=0.5}
  [385] = {accel=40, decel=4000, tmax=21.7, leave=0, reach=0.5}
  [386] = {accel=40, decel=4000, tmax=21.817, leave=0, reach=0.5}
  [387] = {accel=40, decel=4000, tmax=21.917, leave=0, reach=0.5}
  [388] = {accel=40, decel=4000, tmax=21.981, leave=0, reach=0.5}
  [389] = {accel=40, decel=4000, tmax=22.015, leave=0, reach=0.5}
  [390] = {accel=40, decel=4000, tmax=22.04, leave=0, reach=0.5}
  [391] = {accel=40, decel=4000, tmax=22.076, leave=0, reach=0.5}
  [392] = {accel=40, decel=4000, tmax=22.124, leave=0, reach=0.5}
  [393] = {accel=40, decel=4000, tmax=22.169, leave=0, reach=0.5}
  [394] = {accel=40, decel=4000, tmax=22.191, leave=0, reach=0.5}
  [395] = {accel=40, decel=4000, tmax=22.176, leave=0, reach=0.5}
  [396] = {accel=40, decel=4000, tmax=22.123, leave=0, reach=0.5}
  [397] = {accel=40, decel=4000, tmax=22.051, leave=0, reach=0.5}
  [398] = {accel=40, decel=4000, tmax=21.974, leave=0, reach=0.5}
  [399] = {accel=40, decel=4000, tmax=21.898, leave=0, reach=0.5}
  [400] = {accel=40, decel=4000, tmax=21.819, leave=0, reach=0.5}
  [401] = {accel=40, decel=4000, tmax=21.724, leave=0, reach=0.5}
  [402] = {accel=40, decel=4000, tmax=21.607, leave=0, reach=0.5}
  [403] = {accel=40, decel=4000, tmax=21.468, leave=0, reach=0.5}
  [404] = {accel=40, decel=4000, tmax=21.313, leave=0, reach=0.5}
  [405] = {accel=40, decel=4000, tmax=21.147, leave=0, reach=0.5}
  [406] = {accel=40, decel=4000, tmax=20.971, leave=0, reach=0.5}
  [407] = {accel=40, decel=4000, tmax=20.78, leave=0, reach=0.5}
  [408] = {accel=40, decel=4000, tmax=20.572, leave=0, reach=0.5}
  [409] = {accel=40, decel=4000, tmax=20.348, leave=0, reach=0.5}
  [410] = {accel=40, decel=4000, tmax=20.113, leave=0, reach=0.5}
  [411] = {accel=40, decel=4000, tmax=19.87, leave=0, reach=0.5}
  [412] = {accel=40, decel=4000, tmax=19.62, leave=0, reach=0.5}
  [413] = {accel=40, decel=4000, tmax=19.36, leave=0, reach=0.5}
  [414] = {accel=40, decel=4000, tmax=19.09, leave=0, reach=0.5}
  [415] = {accel=40, decel=4000, tmax=18.803, leave=0, reach=0.5}
  [416] = {accel=40, decel=4000, tmax=18.496, leave=0, reach=0.5}
  [417] = {accel=40, decel=4000, tmax=18.158, leave=0, reach=0.5}
  [418] = {accel=40, decel=4000, tmax=17.785, leave=0, reach=0.5}
  [419] = {accel=40, decel=4000, tmax=17.38, leave=0, reach=0.5}
  [420] = {accel=40, decel=4000, tmax=16.952, leave=0, reach=0.5}
  [421] = {accel=40, decel=4000, tmax=16.512, leave=0, reach=0.5}
  [422] = {accel=40, decel=4000, tmax=16.064, leave=0, reach=0.5}
  [423] = {accel=40, decel=4000, tmax=15.613, leave=0, reach=0.5}
  [424] = {accel=40, decel=4000, tmax=15.163, leave=0, reach=0.5}
  [425] = {accel=40, decel=4000, tmax=14.719, leave=0, reach=0.5}
  [426] = {accel=40, decel=4000, tmax=14.289, leave=0, reach=0.5}
  [427] = {accel=40, decel=4000, tmax=13.875, leave=0, reach=0.5}
  [428] = {accel=40, decel=4000, tmax=13.477, leave=0, reach=0.5}
  [429] = {accel=40, decel=4000, tmax=42.678, leave=0, reach=0.5}
  [430] = {accel=40, decel=4000, tmax=13.946, leave=0, reach=0.5}
  [431] = {accel=40, decel=4000, tmax=14.383, leave=0, reach=0.5}
  [432] = {accel=40, decel=4000, tmax=14.831, leave=0, reach=0.5}
  [433] = {accel=40, decel=4000, tmax=15.283, leave=0, reach=0.5}
  [434] = {accel=40, decel=4000, tmax=15.737, leave=0, reach=0.5}
  [435] = {accel=40, decel=4000, tmax=16.189, leave=0, reach=0.5}
  [436] = {accel=40, decel=4000, tmax=16.631, leave=0, reach=0.5}
  [437] = {accel=40, decel=4000, tmax=17.053, leave=0, reach=0.5}
  [438] = {accel=40, decel=4000, tmax=17.441, leave=0, reach=0.5}
  [439] = {accel=40, decel=4000, tmax=17.788, leave=0, reach=0.5}
  [440] = {accel=40, decel=4000, tmax=18.099, leave=0, reach=0.5}
  [441] = {accel=40, decel=4000, tmax=18.388, leave=0, reach=0.5}
  [442] = {accel=40, decel=4000, tmax=18.664, leave=0, reach=0.5}
  [443] = {accel=40, decel=4000, tmax=18.934, leave=0, reach=0.5}
  [444] = {accel=40, decel=4000, tmax=19.198, leave=0, reach=0.5}
  [445] = {accel=40, decel=4000, tmax=19.457, leave=0, reach=0.5}
  [446] = {accel=40, decel=4000, tmax=19.708, leave=0, reach=0.5}
  [447] = {accel=40, decel=4000, tmax=19.949, leave=0, reach=0.5}
  [448] = {accel=40, decel=4000, tmax=20.174, leave=0, reach=0.5}
  [449] = {accel=40, decel=4000, tmax=20.38, leave=0, reach=0.5}
  [450] = {accel=40, decel=4000, tmax=20.572, leave=0, reach=0.5}
  [451] = {accel=40, decel=4000, tmax=20.755, leave=0, reach=0.5}
  [452] = {accel=40, decel=4000, tmax=20.925, leave=0, reach=0.5}
  [453] = {accel=40, decel=4000, tmax=21.073, leave=0, reach=0.5}
  [454] = {accel=40, decel=4000, tmax=21.193, leave=0, reach=0.5}
  [455] = {accel=40, decel=4000, tmax=21.282, leave=0, reach=0.5}
  [456] = {accel=40, decel=4000, tmax=21.354, leave=0, reach=0.5}
  [457] = {accel=40, decel=4000, tmax=21.424, leave=0, reach=0.5}
  [458] = {accel=40, decel=4000, tmax=21.506, leave=0, reach=0.5}
  [459] = {accel=40, decel=4000, tmax=21.594, leave=0, reach=0.5}
  [460] = {accel=40, decel=4000, tmax=21.669, leave=0, reach=0.5}
  [461] = {accel=40, decel=4000, tmax=21.706, leave=0, reach=0.5}
  [462] = {accel=40, decel=4000, tmax=21.693, leave=0, reach=0.5}
  [463] = {accel=40, decel=4000, tmax=21.642, leave=0, reach=0.5}
  [464] = {accel=40, decel=4000, tmax=21.578, leave=0, reach=0.5}
  [465] = {accel=40, decel=4000, tmax=21.526, leave=0, reach=0.5}
  [466] = {accel=40, decel=4000, tmax=21.496, leave=0, reach=0.5}
  [467] = {accel=40, decel=4000, tmax=21.476, leave=0, reach=0.5}
  [468] = {accel=40, decel=4000, tmax=21.442, leave=0, reach=0.5}
  [469] = {accel=40, decel=4000, tmax=21.383, leave=0, reach=0.5}
  [470] = {accel=40, decel=4000, tmax=21.306, leave=0, reach=0.5}
  [471] = {accel=40, decel=4000, tmax=21.233, leave=0, reach=0.5}
  [472] = {accel=40, decel=4000, tmax=21.186, leave=0, reach=0.5}
  [473] = {accel=40, decel=4000, tmax=21.172, leave=0, reach=0.5}
  [474] = {accel=40, decel=4000, tmax=21.183, leave=0, reach=0.5}
  [475] = {accel=40, decel=4000, tmax=21.203, leave=0, reach=0.5}
  [476] = {accel=40, decel=4000, tmax=21.221, leave=0, reach=0.5}
  [477] = {accel=40, decel=4000, tmax=21.232, leave=0, reach=0.5}
  [478] = {accel=40, decel=4000, tmax=21.239, leave=0, reach=0.5}
  [479] = {accel=40, decel=4000, tmax=21.245, leave=0, reach=0.5}
  [480] = {accel=40, decel=4000, tmax=21.252, leave=0, reach=0.5}
  [481] = {accel=40, decel=4000, tmax=21.261, leave=0, reach=0.5}
  [482] = {accel=40, decel=4000, tmax=21.258, leave=0, reach=0.5}
  [483] = {accel=40, decel=4000, tmax=21.229, leave=0, reach=0.5}
  [484] = {accel=40, decel=4000, tmax=21.159, leave=0, reach=0.5}
  [485] = {accel=40, decel=4000, tmax=21.042, leave=0, reach=0.5}
  [486] = {accel=40, decel=4000, tmax=20.886, leave=0, reach=0.5}
  [487] = {accel=40, decel=4000, tmax=20.702, leave=0, reach=0.5}
  [488] = {accel=40, decel=4000, tmax=20.501, leave=0, reach=0.5}
  [489] = {accel=40, decel=4000, tmax=20.287, leave=0, reach=0.5}
  [490] = {accel=40, decel=4000, tmax=20.058, leave=0, reach=0.5}
  [491] = {accel=40, decel=4000, tmax=19.806, leave=0, reach=0.5}
  [492] = {accel=40, decel=4000, tmax=19.519, leave=0, reach=0.5}
  [493] = {accel=40, decel=4000, tmax=19.194, leave=0, reach=0.5}
  [494] = {accel=40, decel=4000, tmax=18.837, leave=0, reach=0.5}
  [495] = {accel=40, decel=4000, tmax=18.459, leave=0, reach=0.5}
  [496] = {accel=40, decel=4000, tmax=18.068, leave=0, reach=0.5}
  [497] = {accel=40, decel=4000, tmax=17.668, leave=0, reach=0.5}
  [498] = {accel=40, decel=4000, tmax=17.255, leave=0, reach=0.5}
  [499] = {accel=40, decel=4000, tmax=16.829, leave=0, reach=0.5}
  [500] = {accel=40, decel=4000, tmax=16.388, leave=0, reach=0.5}
  [501] = {accel=40, decel=4000, tmax=15.928, leave=0, reach=0.5}
  [502] = {accel=40, decel=4000, tmax=34.908, leave=0, reach=0.5}
  [503] = {accel=40, decel=4000, tmax=15.769, leave=0, reach=0.5}
  [504] = {accel=40, decel=4000, tmax=16.217, leave=0, reach=0.5}
  [505] = {accel=40, decel=4000, tmax=16.654, leave=0, reach=0.5}
  [506] = {accel=40, decel=4000, tmax=17.082, leave=0, reach=0.5}
  [507] = {accel=40, decel=4000, tmax=17.499, leave=0, reach=0.5}
  [508] = {accel=40, decel=4000, tmax=17.904, leave=0, reach=0.5}
  [509] = {accel=40, decel=4000, tmax=18.294, leave=0, reach=0.5}
  [510] = {accel=40, decel=4000, tmax=18.659, leave=0, reach=0.5}
  [511] = {accel=40, decel=4000, tmax=19.004, leave=0, reach=0.5}
  [512] = {accel=40, decel=4000, tmax=19.333, leave=0, reach=0.5}
  [513] = {accel=40, decel=4000, tmax=19.64, leave=0, reach=0.5}
  [514] = {accel=40, decel=4000, tmax=19.921, leave=0, reach=0.5}
  [515] = {accel=40, decel=4000, tmax=20.178, leave=0, reach=0.5}
  [516] = {accel=40, decel=4000, tmax=20.409, leave=0, reach=0.5}
  [517] = {accel=40, decel=4000, tmax=20.607, leave=0, reach=0.5}
  [518] = {accel=40, decel=4000, tmax=20.758, leave=0, reach=0.5}
  [519] = {accel=40, decel=4000, tmax=20.854, leave=0, reach=0.5}
  [520] = {accel=40, decel=4000, tmax=20.9, leave=0, reach=0.5}
  [521] = {accel=40, decel=4000, tmax=20.913, leave=0, reach=0.5}
  [522] = {accel=40, decel=4000, tmax=20.91, leave=0, reach=0.5}
  [523] = {accel=40, decel=4000, tmax=20.907, leave=0, reach=0.5}
  [524] = {accel=40, decel=4000, tmax=20.904, leave=0, reach=0.5}
  [525] = {accel=40, decel=4000, tmax=20.904, leave=0, reach=0.5}
  [526] = {accel=40, decel=4000, tmax=20.906, leave=0, reach=0.5}
  [527] = {accel=40, decel=4000, tmax=20.886, leave=0, reach=0.5}
  [528] = {accel=40, decel=4000, tmax=20.858, leave=0, reach=0.5}
  [529] = {accel=40, decel=4000, tmax=20.843, leave=0, reach=0.5}
  [530] = {accel=40, decel=4000, tmax=20.83, leave=0, reach=0.5}
  [531] = {accel=40, decel=4000, tmax=20.836, leave=0, reach=0.5}
  [532] = {accel=40, decel=4000, tmax=20.87, leave=0, reach=0.5}
  [533] = {accel=40, decel=4000, tmax=20.912, leave=0, reach=0.5}
  [534] = {accel=40, decel=4000, tmax=20.947, leave=0, reach=0.5}
  [535] = {accel=40, decel=4000, tmax=20.969, leave=0, reach=0.5}
  [536] = {accel=40, decel=4000, tmax=20.992, leave=0, reach=0.5}
  [537] = {accel=40, decel=4000, tmax=21.043, leave=0, reach=0.5}
  [538] = {accel=40, decel=4000, tmax=21.126, leave=0, reach=0.5}
  [539] = {accel=40, decel=4000, tmax=21.214, leave=0, reach=0.5}
  [540] = {accel=40, decel=4000, tmax=21.271, leave=0, reach=0.5}
  [541] = {accel=40, decel=4000, tmax=21.272, leave=0, reach=0.5}
  [542] = {accel=40, decel=4000, tmax=21.214, leave=0, reach=0.5}
  [543] = {accel=40, decel=4000, tmax=21.119, leave=0, reach=0.5}
  [544] = {accel=40, decel=4000, tmax=21.008, leave=0, reach=0.5}
  [545] = {accel=40, decel=4000, tmax=20.897, leave=0, reach=0.5}
  [546] = {accel=40, decel=4000, tmax=20.816, leave=0, reach=0.5}
  [547] = {accel=40, decel=4000, tmax=20.737, leave=0, reach=0.5}
  [548] = {accel=40, decel=4000, tmax=20.627, leave=0, reach=0.5}
  [549] = {accel=40, decel=4000, tmax=20.489, leave=0, reach=0.5}
  [550] = {accel=40, decel=4000, tmax=20.316, leave=0, reach=0.5}
  [551] = {accel=40, decel=4000, tmax=20.118, leave=0, reach=0.5}
  [552] = {accel=40, decel=4000, tmax=19.914, leave=0, reach=0.5}
  [553] = {accel=40, decel=4000, tmax=19.705, leave=0, reach=0.5}
  [554] = {accel=40, decel=4000, tmax=19.487, leave=0, reach=0.5}
  [555] = {accel=40, decel=4000, tmax=19.249, leave=0, reach=0.5}
  [556] = {accel=40, decel=4000, tmax=18.991, leave=0, reach=0.5}
  [557] = {accel=40, decel=4000, tmax=18.716, leave=0, reach=0.5}
  [558] = {accel=40, decel=4000, tmax=18.434, leave=0, reach=0.5}
  [559] = {accel=40, decel=4000, tmax=18.149, leave=0, reach=0.5}
  [560] = {accel=40, decel=4000, tmax=17.859, leave=0, reach=0.5}
  [561] = {accel=40, decel=4000, tmax=17.563, leave=0, reach=0.5}
  [562] = {accel=40, decel=4000, tmax=17.254, leave=0, reach=0.5}
  [563] = {accel=40, decel=4000, tmax=16.929, leave=0, reach=0.5}
  [564] = {accel=40, decel=4000, tmax=16.575, leave=0, reach=0.5}
  [565] = {accel=40, decel=4000, tmax=16.178, leave=0, reach=0.5}
  [566] = {accel=40, decel=4000, tmax=15.748, leave=0, reach=0.5}
  [567] = {accel=40, decel=4000, tmax=15.304, leave=0, reach=0.5}
  [568] = {accel=40, decel=4000, tmax=14.859, leave=0, reach=0.5}
  [569] = {accel=40, decel=4000, tmax=14.42, leave=0, reach=0.5}
  [570] = {accel=40, decel=4000, tmax=13.991, leave=0, reach=0.5}
  [571] = {accel=40, decel=4000, tmax=44.09, leave=0, reach=0.5}
  [572] = {accel=40, decel=4000, tmax=14.331, leave=0, reach=0.5}
  [573] = {accel=40, decel=4000, tmax=14.754, leave=0, reach=0.5}
  [574] = {accel=40, decel=4000, tmax=15.171, leave=0, reach=0.5}
  [575] = {accel=40, decel=4000, tmax=15.563, leave=0, reach=0.5}
  [576] = {accel=40, decel=4000, tmax=15.919, leave=0, reach=0.5}
  [577] = {accel=40, decel=4000, tmax=16.246, leave=0, reach=0.5}
  [578] = {accel=40, decel=4000, tmax=16.558, leave=0, reach=0.5}
  [579] = {accel=40, decel=4000, tmax=16.858, leave=0, reach=0.5}
  [580] = {accel=40, decel=4000, tmax=17.154, leave=0, reach=0.5}
  [581] = {accel=40, decel=4000, tmax=17.446, leave=0, reach=0.5}
  [582] = {accel=40, decel=4000, tmax=17.73, leave=0, reach=0.5}
  [583] = {accel=40, decel=4000, tmax=18.002, leave=0, reach=0.5}
  [584] = {accel=40, decel=4000, tmax=18.256, leave=0, reach=0.5}
  [585] = {accel=40, decel=4000, tmax=18.484, leave=0, reach=0.5}
  [586] = {accel=40, decel=4000, tmax=18.69, leave=0, reach=0.5}
  [587] = {accel=40, decel=4000, tmax=18.893, leave=0, reach=0.5}
  [588] = {accel=40, decel=4000, tmax=19.103, leave=0, reach=0.5}
  [589] = {accel=40, decel=4000, tmax=19.317, leave=0, reach=0.5}
  [590] = {accel=40, decel=4000, tmax=19.521, leave=0, reach=0.5}
  [591] = {accel=40, decel=4000, tmax=19.696, leave=0, reach=0.5}
  [592] = {accel=40, decel=4000, tmax=19.835, leave=0, reach=0.5}
  [593] = {accel=40, decel=4000, tmax=19.953, leave=0, reach=0.5}
  [594] = {accel=40, decel=4000, tmax=20.079, leave=0, reach=0.5}
  [595] = {accel=40, decel=4000, tmax=20.224, leave=0, reach=0.5}
  [596] = {accel=40, decel=4000, tmax=20.375, leave=0, reach=0.5}
  [597] = {accel=40, decel=4000, tmax=20.509, leave=0, reach=0.5}
  [598] = {accel=40, decel=4000, tmax=20.594, leave=0, reach=0.5}
  [599] = {accel=40, decel=4000, tmax=20.605, leave=0, reach=0.5}
  [600] = {accel=40, decel=4000, tmax=20.546, leave=0, reach=0.5}
  [601] = {accel=40, decel=4000, tmax=20.445, leave=0, reach=0.5}
  [602] = {accel=40, decel=4000, tmax=20.343, leave=0, reach=0.5}
  [603] = {accel=40, decel=4000, tmax=20.266, leave=0, reach=0.5}
  [604] = {accel=40, decel=4000, tmax=20.221, leave=0, reach=0.5}
  [605] = {accel=40, decel=4000, tmax=20.193, leave=0, reach=0.5}
  [606] = {accel=40, decel=4000, tmax=20.168, leave=0, reach=0.5}
  [607] = {accel=40, decel=4000, tmax=20.148, leave=0, reach=0.5}
  [608] = {accel=40, decel=4000, tmax=20.139, leave=0, reach=0.5}
  [609] = {accel=40, decel=4000, tmax=20.142, leave=0, reach=0.5}
  [610] = {accel=40, decel=4000, tmax=20.153, leave=0, reach=0.5}
  [611] = {accel=40, decel=4000, tmax=20.172, leave=0, reach=0.5}
  [612] = {accel=40, decel=4000, tmax=20.192, leave=0, reach=0.5}
  [613] = {accel=40, decel=4000, tmax=20.199, leave=0, reach=0.5}
  [614] = {accel=40, decel=4000, tmax=20.193, leave=0, reach=0.5}
  [615] = {accel=40, decel=4000, tmax=20.184, leave=0, reach=0.5}
  [616] = {accel=40, decel=4000, tmax=20.18, leave=0, reach=0.5}
  [617] = {accel=40, decel=4000, tmax=20.183, leave=0, reach=0.5}
  [618] = {accel=40, decel=4000, tmax=20.184, leave=0, reach=0.5}
  [619] = {accel=40, decel=4000, tmax=20.166, leave=0, reach=0.5}
  [620] = {accel=40, decel=4000, tmax=20.112, leave=0, reach=0.5}
  [621] = {accel=40, decel=4000, tmax=20.005, leave=0, reach=0.5}
  [622] = {accel=40, decel=4000, tmax=19.84, leave=0, reach=0.5}
  [623] = {accel=40, decel=4000, tmax=19.625, leave=0, reach=0.5}
  [624] = {accel=40, decel=4000, tmax=19.372, leave=0, reach=0.5}
  [625] = {accel=40, decel=4000, tmax=19.081, leave=0, reach=0.5}
  [626] = {accel=40, decel=4000, tmax=18.756, leave=0, reach=0.5}
  [627] = {accel=40, decel=4000, tmax=18.402, leave=0, reach=0.5}
  [628] = {accel=40, decel=4000, tmax=18.028, leave=0, reach=0.5}
  [629] = {accel=40, decel=4000, tmax=17.645, leave=0, reach=0.5}
  [630] = {accel=40, decel=4000, tmax=17.251, leave=0, reach=0.5}
  [631] = {accel=40, decel=4000, tmax=16.841, leave=0, reach=0.5}
  [632] = {accel=40, decel=4000, tmax=16.419, leave=0, reach=0.5}
  [633] = {accel=40, decel=4000, tmax=15.989, leave=0, reach=0.5}
  [634] = {accel=40, decel=4000, tmax=50.047, leave=0, reach=0.5}
  [635] = {accel=40, decel=4000, tmax=16.094, leave=0, reach=0.5}
  [636] = {accel=40, decel=4000, tmax=16.498, leave=0, reach=0.5}
  [637] = {accel=40, decel=4000, tmax=16.896, leave=0, reach=0.5}
  [638] = {accel=40, decel=4000, tmax=17.288, leave=0, reach=0.5}
  [639] = {accel=40, decel=4000, tmax=17.663, leave=0, reach=0.5}
  [640] = {accel=40, decel=4000, tmax=18.009, leave=0, reach=0.5}
  [641] = {accel=40, decel=4000, tmax=18.32, leave=0, reach=0.5}
  [642] = {accel=40, decel=4000, tmax=18.588, leave=0, reach=0.5}
  [643] = {accel=40, decel=4000, tmax=18.81, leave=0, reach=0.5}
  [644] = {accel=40, decel=4000, tmax=18.982, leave=0, reach=0.5}
  [645] = {accel=40, decel=4000, tmax=19.094, leave=0, reach=0.5}
  [646] = {accel=40, decel=4000, tmax=19.158, leave=0, reach=0.5}
  [647] = {accel=40, decel=4000, tmax=19.194, leave=0, reach=0.5}
  [648] = {accel=40, decel=4000, tmax=19.212, leave=0, reach=0.5}
  [649] = {accel=40, decel=4000, tmax=19.221, leave=0, reach=0.5}
  [650] = {accel=40, decel=4000, tmax=19.226, leave=0, reach=0.5}
  [651] = {accel=40, decel=4000, tmax=19.226, leave=0, reach=0.5}
  [652] = {accel=40, decel=4000, tmax=19.218, leave=0, reach=0.5}
  [653] = {accel=40, decel=4000, tmax=19.196, leave=0, reach=0.5}
  [654] = {accel=40, decel=4000, tmax=19.168, leave=0, reach=0.5}
  [655] = {accel=40, decel=4000, tmax=19.148, leave=0, reach=0.5}
  [656] = {accel=40, decel=4000, tmax=19.143, leave=0, reach=0.5}
  [657] = {accel=40, decel=4000, tmax=19.152, leave=0, reach=0.5}
  [658] = {accel=40, decel=4000, tmax=19.174, leave=0, reach=0.5}
  [659] = {accel=40, decel=4000, tmax=19.204, leave=0, reach=0.5}
  [660] = {accel=40, decel=4000, tmax=19.239, leave=0, reach=0.5}
  [661] = {accel=40, decel=4000, tmax=19.282, leave=0, reach=0.5}
  [662] = {accel=40, decel=4000, tmax=19.342, leave=0, reach=0.5}
  [663] = {accel=40, decel=4000, tmax=19.425, leave=0, reach=0.5}
  [664] = {accel=40, decel=4000, tmax=19.531, leave=0, reach=0.5}
  [665] = {accel=40, decel=4000, tmax=19.629, leave=0, reach=0.5}
  [666] = {accel=40, decel=4000, tmax=19.676, leave=0, reach=0.5}
  [667] = {accel=40, decel=4000, tmax=19.645, leave=0, reach=0.5}
  [668] = {accel=40, decel=4000, tmax=19.539, leave=0, reach=0.5}
  [669] = {accel=40, decel=4000, tmax=19.382, leave=0, reach=0.5}
  [670] = {accel=40, decel=4000, tmax=19.201, leave=0, reach=0.5}
  [671] = {accel=40, decel=4000, tmax=19.02, leave=0, reach=0.5}
  [672] = {accel=40, decel=4000, tmax=18.856, leave=0, reach=0.5}
  [673] = {accel=40, decel=4000, tmax=18.698, leave=0, reach=0.5}
  [674] = {accel=40, decel=4000, tmax=18.524, leave=0, reach=0.5}
  [675] = {accel=40, decel=4000, tmax=18.319, leave=0, reach=0.5}
  [676] = {accel=40, decel=4000, tmax=18.089, leave=0, reach=0.5}
  [677] = {accel=40, decel=4000, tmax=17.854, leave=0, reach=0.5}
  [678] = {accel=40, decel=4000, tmax=17.632, leave=0, reach=0.5}
  [679] = {accel=40, decel=4000, tmax=17.431, leave=0, reach=0.5}
  [680] = {accel=40, decel=4000, tmax=17.24, leave=0, reach=0.5}
  [681] = {accel=40, decel=4000, tmax=17.035, leave=0, reach=0.5}
  [682] = {accel=40, decel=4000, tmax=16.802, leave=0, reach=0.5}
  [683] = {accel=40, decel=4000, tmax=16.542, leave=0, reach=0.5}
  [684] = {accel=40, decel=4000, tmax=16.262, leave=0, reach=0.5}
  [685] = {accel=40, decel=4000, tmax=15.973, leave=0, reach=0.5}
  [686] = {accel=40, decel=4000, tmax=15.684, leave=0, reach=0.5}
  [687] = {accel=40, decel=4000, tmax=15.393, leave=0, reach=0.5}
  [688] = {accel=40, decel=4000, tmax=15.096, leave=0, reach=0.5}
  [689] = {accel=40, decel=4000, tmax=14.783, leave=0, reach=0.5}
  [690] = {accel=40, decel=4000, tmax=14.446, leave=0, reach=0.5}
  [691] = {accel=40, decel=4000, tmax=44.945, leave=0, reach=0.5}
  [692] = {accel=40, decel=4000, tmax=14.295, leave=0, reach=0.5}
  [693] = {accel=40, decel=4000, tmax=14.561, leave=0, reach=0.5}
  [694] = {accel=40, decel=4000, tmax=14.832, leave=0, reach=0.5}
  [695] = {accel=40, decel=4000, tmax=15.107, leave=0, reach=0.5}
  [696] = {accel=40, decel=4000, tmax=15.376, leave=0, reach=0.5}
  [697] = {accel=40, decel=4000, tmax=15.624, leave=0, reach=0.5}
  [698] = {accel=40, decel=4000, tmax=15.841, leave=0, reach=0.5}
  [699] = {accel=40, decel=4000, tmax=16.038, leave=0, reach=0.5}
  [700] = {accel=40, decel=4000, tmax=16.233, leave=0, reach=0.5}
  [701] = {accel=40, decel=4000, tmax=16.439, leave=0, reach=0.5}
  [702] = {accel=40, decel=4000, tmax=16.665, leave=0, reach=0.5}
  [703] = {accel=40, decel=4000, tmax=16.906, leave=0, reach=0.5}
  [704] = {accel=40, decel=4000, tmax=17.148, leave=0, reach=0.5}
  [705] = {accel=40, decel=4000, tmax=17.373, leave=0, reach=0.5}
  [706] = {accel=40, decel=4000, tmax=17.576, leave=0, reach=0.5}
  [707] = {accel=40, decel=4000, tmax=17.766, leave=0, reach=0.5}
  [708] = {accel=40, decel=4000, tmax=17.96, leave=0, reach=0.5}
  [709] = {accel=40, decel=4000, tmax=18.161, leave=0, reach=0.5}
  [710] = {accel=40, decel=4000, tmax=18.351, leave=0, reach=0.5}
  [711] = {accel=40, decel=4000, tmax=18.505, leave=0, reach=0.5}
  [712] = {accel=40, decel=4000, tmax=18.604, leave=0, reach=0.5}
  [713] = {accel=40, decel=4000, tmax=18.637, leave=0, reach=0.5}
  [714] = {accel=40, decel=4000, tmax=18.607, leave=0, reach=0.5}
  [715] = {accel=40, decel=4000, tmax=18.539, leave=0, reach=0.5}
  [716] = {accel=40, decel=4000, tmax=18.456, leave=0, reach=0.5}
  [717] = {accel=40, decel=4000, tmax=18.375, leave=0, reach=0.5}
  [718] = {accel=40, decel=4000, tmax=18.302, leave=0, reach=0.5}
  [719] = {accel=40, decel=4000, tmax=18.237, leave=0, reach=0.5}
  [720] = {accel=40, decel=4000, tmax=18.179, leave=0, reach=0.5}
  [721] = {accel=40, decel=4000, tmax=18.126, leave=0, reach=0.5}
  [722] = {accel=40, decel=4000, tmax=18.08, leave=0, reach=0.5}
  [723] = {accel=40, decel=4000, tmax=18.046, leave=0, reach=0.5}
  [724] = {accel=40, decel=4000, tmax=18.037, leave=0, reach=0.5}
  [725] = {accel=40, decel=4000, tmax=18.063, leave=0, reach=0.5}
  [726] = {accel=40, decel=4000, tmax=18.114, leave=0, reach=0.5}
  [727] = {accel=40, decel=4000, tmax=18.169, leave=0, reach=0.5}
  [728] = {accel=40, decel=4000, tmax=18.211, leave=0, reach=0.5}
  [729] = {accel=40, decel=4000, tmax=18.235, leave=0, reach=0.5}
  [730] = {accel=40, decel=4000, tmax=18.242, leave=0, reach=0.5}
  [731] = {accel=40, decel=4000, tmax=18.231, leave=0, reach=0.5}
  [732] = {accel=40, decel=4000, tmax=18.198, leave=0, reach=0.5}
  [733] = {accel=40, decel=4000, tmax=18.139, leave=0, reach=0.5}
  [734] = {accel=40, decel=4000, tmax=18.044, leave=0, reach=0.5}
  [735] = {accel=40, decel=4000, tmax=17.907, leave=0, reach=0.5}
  [736] = {accel=40, decel=4000, tmax=17.726, leave=0, reach=0.5}
  [737] = {accel=40, decel=4000, tmax=17.494, leave=0, reach=0.5}
  [738] = {accel=40, decel=4000, tmax=17.214, leave=0, reach=0.5}
  [739] = {accel=40, decel=4000, tmax=16.895, leave=0, reach=0.5}
  [740] = {accel=40, decel=4000, tmax=16.544, leave=0, reach=0.5}
  [741] = {accel=40, decel=4000, tmax=67.623, leave=0, reach=0.5}
  [742] = {accel=40, decel=4000, tmax=16.557, leave=0, reach=0.5}
  [743] = {accel=40, decel=4000, tmax=16.76, leave=0, reach=0.5}
  [744] = {accel=40, decel=4000, tmax=16.925, leave=0, reach=0.5}
  [745] = {accel=40, decel=4000, tmax=17.046, leave=0, reach=0.5}
  [746] = {accel=40, decel=4000, tmax=17.125, leave=0, reach=0.5}
  [747] = {accel=40, decel=4000, tmax=17.165, leave=0, reach=0.5}
  [748] = {accel=40, decel=4000, tmax=17.171, leave=0, reach=0.5}
  [749] = {accel=40, decel=4000, tmax=17.144, leave=0, reach=0.5}
  [750] = {accel=40, decel=4000, tmax=17.087, leave=0, reach=0.5}
  [751] = {accel=40, decel=4000, tmax=17.008, leave=0, reach=0.5}
  [752] = {accel=40, decel=4000, tmax=16.92, leave=0, reach=0.5}
  [753] = {accel=40, decel=4000, tmax=16.845, leave=0, reach=0.5}
  [754] = {accel=40, decel=4000, tmax=16.813, leave=0, reach=0.5}
  [755] = {accel=40, decel=4000, tmax=16.834, leave=0, reach=0.5}
  [756] = {accel=40, decel=4000, tmax=16.897, leave=0, reach=0.5}
  [757] = {accel=40, decel=4000, tmax=16.98, leave=0, reach=0.5}
  [758] = {accel=40, decel=4000, tmax=17.064, leave=0, reach=0.5}
  [759] = {accel=40, decel=4000, tmax=17.146, leave=0, reach=0.5}
  [760] = {accel=40, decel=4000, tmax=17.231, leave=0, reach=0.5}
  [761] = {accel=40, decel=4000, tmax=17.314, leave=0, reach=0.5}
  [762] = {accel=40, decel=4000, tmax=17.385, leave=0, reach=0.5}
  [763] = {accel=40, decel=4000, tmax=17.438, leave=0, reach=0.5}
  [764] = {accel=40, decel=4000, tmax=17.472, leave=0, reach=0.5}
  [765] = {accel=40, decel=4000, tmax=17.478, leave=0, reach=0.5}
  [766] = {accel=40, decel=4000, tmax=17.442, leave=0, reach=0.5}
  [767] = {accel=40, decel=4000, tmax=17.359, leave=0, reach=0.5}
  [768] = {accel=40, decel=4000, tmax=17.227, leave=0, reach=0.5}
  [769] = {accel=40, decel=4000, tmax=17.053, leave=0, reach=0.5}
  [770] = {accel=40, decel=4000, tmax=16.852, leave=0, reach=0.5}
  [771] = {accel=40, decel=4000, tmax=16.643, leave=0, reach=0.5}
  [772] = {accel=40, decel=4000, tmax=16.431, leave=0, reach=0.5}
  [773] = {accel=40, decel=4000, tmax=16.211, leave=0, reach=0.5}
  [774] = {accel=40, decel=4000, tmax=15.978, leave=0, reach=0.5}
  [775] = {accel=40, decel=4000, tmax=15.737, leave=0, reach=0.5}
  [776] = {accel=40, decel=4000, tmax=15.499, leave=0, reach=0.5}
  [777] = {accel=40, decel=4000, tmax=15.274, leave=0, reach=0.5}
  [778] = {accel=40, decel=4000, tmax=15.065, leave=0, reach=0.5}
  [779] = {accel=40, decel=4000, tmax=14.867, leave=0, reach=0.5}
  [780] = {accel=40, decel=4000, tmax=14.665, leave=0, reach=0.5}
  [781] = {accel=40, decel=4000, tmax=14.449, leave=0, reach=0.5}
  [782] = {accel=40, decel=4000, tmax=14.217, leave=0, reach=0.5}
  [783] = {accel=40, decel=4000, tmax=71.934, leave=0, reach=0.5}
  [784] = {accel=40, decel=4000, tmax=14.23, leave=0, reach=0.5}
  [785] = {accel=40, decel=4000, tmax=14.452, leave=0, reach=0.5}
  [786] = {accel=40, decel=4000, tmax=14.685, leave=0, reach=0.5}
  [787] = {accel=40, decel=4000, tmax=14.922, leave=0, reach=0.5}
  [788] = {accel=40, decel=4000, tmax=15.158, leave=0, reach=0.5}
  [789] = {accel=40, decel=4000, tmax=15.391, leave=0, reach=0.5}
  [790] = {accel=40, decel=4000, tmax=15.612, leave=0, reach=0.5}
  [791] = {accel=40, decel=4000, tmax=15.822, leave=0, reach=0.5}
  [792] = {accel=40, decel=4000, tmax=16.017, leave=0, reach=0.5}
  [793] = {accel=40, decel=4000, tmax=16.167, leave=0, reach=0.5}
  [794] = {accel=40, decel=4000, tmax=16.269, leave=0, reach=0.5}
  [795] = {accel=40, decel=4000, tmax=16.341, leave=0, reach=0.5}
  [796] = {accel=40, decel=4000, tmax=16.389, leave=0, reach=0.5}
  [797] = {accel=40, decel=4000, tmax=16.413, leave=0, reach=0.5}
  [798] = {accel=40, decel=4000, tmax=16.41, leave=0, reach=0.5}
  [799] = {accel=40, decel=4000, tmax=16.374, leave=0, reach=0.5}
  [800] = {accel=40, decel=4000, tmax=16.314, leave=0, reach=0.5}
  [801] = {accel=40, decel=4000, tmax=16.236, leave=0, reach=0.5}
  [802] = {accel=40, decel=4000, tmax=16.141, leave=0, reach=0.5}
  [803] = {accel=40, decel=4000, tmax=16.033, leave=0, reach=0.5}
  [804] = {accel=40, decel=4000, tmax=15.916, leave=0, reach=0.5}
  [805] = {accel=40, decel=4000, tmax=15.803, leave=0, reach=0.5}
  [806] = {accel=40, decel=4000, tmax=15.725, leave=0, reach=0.5}
  [807] = {accel=40, decel=4000, tmax=15.695, leave=0, reach=0.5}
  [808] = {accel=40, decel=4000, tmax=15.721, leave=0, reach=0.5}
  [809] = {accel=40, decel=4000, tmax=15.805, leave=0, reach=0.5}
  [810] = {accel=40, decel=4000, tmax=15.91, leave=0, reach=0.5}
  [811] = {accel=40, decel=4000, tmax=16.005, leave=0, reach=0.5}
  [812] = {accel=40, decel=4000, tmax=16.079, leave=0, reach=0.5}
  [813] = {accel=40, decel=4000, tmax=16.118, leave=0, reach=0.5}
  [814] = {accel=40, decel=4000, tmax=16.116, leave=0, reach=0.5}
  [815] = {accel=40, decel=4000, tmax=123.539, leave=0, reach=0.5}
  [816] = {accel=40, decel=4000, tmax=14.653, leave=0, reach=0.5}
  [817] = {accel=40, decel=4000, tmax=14.752, leave=0, reach=0.5}
  [818] = {accel=40, decel=4000, tmax=14.885, leave=0, reach=0.5}
  [819] = {accel=40, decel=4000, tmax=15.028, leave=0, reach=0.5}
  [820] = {accel=40, decel=4000, tmax=15.158, leave=0, reach=0.5}
  [821] = {accel=40, decel=4000, tmax=15.258, leave=0, reach=0.5}
  [822] = {accel=40, decel=4000, tmax=15.331, leave=0, reach=0.5}
  [823] = {accel=40, decel=4000, tmax=15.381, leave=0, reach=0.5}
  [824] = {accel=40, decel=4000, tmax=15.4, leave=0, reach=0.5}
  [825] = {accel=40, decel=4000, tmax=15.381, leave=0, reach=0.5}
  [826] = {accel=40, decel=4000, tmax=15.327, leave=0, reach=0.5}
  [827] = {accel=40, decel=4000, tmax=15.257, leave=0, reach=0.5}
  [828] = {accel=40, decel=4000, tmax=15.177, leave=0, reach=0.5}
  [829] = {accel=40, decel=4000, tmax=15.078, leave=0, reach=0.5}
  [830] = {accel=40, decel=4000, tmax=9.942, leave=0, reach=0.5}
  [831] = {accel=40, decel=4000, tmax=40, leave=0, reach=0.5}
  [832] = {accel=40, decel=4000, tmax=19.17, leave=0.5, reach=0.5}
  [833] = {accel=40, decel=4000, tmax=19.15, leave=0.5, reach=0.5}
  [834] = {accel=40, decel=4000, tmax=19.152, leave=0.5, reach=0.5}
  [835] = {accel=40, decel=4000, tmax=19.17, leave=0.5, reach=0.5}
  [836] = {accel=40, decel=4000, tmax=19.201, leave=0.5, reach=0.5}
  [837] = {accel=40, decel=4000, tmax=19.238, leave=0.5, reach=0.5}
  [838] = {accel=40, decel=4000, tmax=19.273, leave=0.5, reach=0.5}
  [839] = {accel=40, decel=4000, tmax=19.306, leave=0.5, reach=0.5}
  [840] = {accel=40, decel=4000, tmax=19.354, leave=0.5, reach=0.5}
  [841] = {accel=40, decel=4000, tmax=19.43, leave=0.5, reach=0.5}
  [842] = {accel=40, decel=4000, tmax=19.525, leave=0.5, reach=0.5}
  [843] = {accel=40, decel=4000, tmax=19.62, leave=0.5, reach=0.5}
  [844] = {accel=40, decel=4000, tmax=19.71, leave=0.5, reach=0.5}
  [845] = {accel=40, decel=4000, tmax=19.811, leave=0.5, reach=0.5}
  [846] = {accel=40, decel=4000, tmax=19.946, leave=0.5, reach=0.5}
  [847] = {accel=40, decel=4000, tmax=20.124, leave=0.5, reach=0.5}
  [848] = {accel=40, decel=4000, tmax=20.336, leave=0.5, reach=0.5}
  [849] = {accel=40, decel=4000, tmax=20.562, leave=0.5, reach=0.5}
  [850] = {accel=40, decel=4000, tmax=20.776, leave=0.5, reach=0.5}
  [851] = {accel=40, decel=4000, tmax=20.957, leave=0.5, reach=0.5}
  [852] = {accel=40, decel=4000, tmax=21.1, leave=0.5, reach=0.5}
  [853] = {accel=40, decel=4000, tmax=21.21, leave=0.5, reach=0.5}
  [854] = {accel=40, decel=4000, tmax=21.3, leave=0.5, reach=0.5}
  [855] = {accel=40, decel=4000, tmax=21.377, leave=0.5, reach=0.5}
  [856] = {accel=40, decel=4000, tmax=21.436, leave=0.5, reach=0.5}
  [857] = {accel=40, decel=4000, tmax=21.469, leave=0.5, reach=0.5}
  [858] = {accel=40, decel=4000, tmax=21.476, leave=0.5, reach=0.5}
  [859] = {accel=40, decel=4000, tmax=21.468, leave=0.5, reach=0.5}
  [860] = {accel=40, decel=4000, tmax=21.455, leave=0.5, reach=0.5}
  [861] = {accel=40, decel=4000, tmax=21.438, leave=0.5, reach=0.5}
  [862] = {accel=40, decel=4000, tmax=21.414, leave=0.5, reach=0.5}
  [863] = {accel=40, decel=4000, tmax=21.378, leave=0.5, reach=0.5}
  [864] = {accel=40, decel=4000, tmax=21.333, leave=0.5, reach=0.5}
  [865] = {accel=40, decel=4000, tmax=21.287, leave=0.5, reach=0.5}
  [866] = {accel=40, decel=4000, tmax=21.249, leave=0.5, reach=0.5}
  [867] = {accel=40, decel=4000, tmax=21.224, leave=0.5, reach=0.5}
  [868] = {accel=40, decel=4000, tmax=21.207, leave=0.5, reach=0.5}
  [869] = {accel=40, decel=4000, tmax=21.191, leave=0.5, reach=0.5}
  [870] = {accel=40, decel=4000, tmax=21.167, leave=0.5, reach=0.5}
  [871] = {accel=40, decel=4000, tmax=21.132, leave=0.5, reach=0.5}
  [872] = {accel=40, decel=4000, tmax=21.081, leave=0.5, reach=0.5}
  [873] = {accel=40, decel=4000, tmax=21.01, leave=0.5, reach=0.5}
  [874] = {accel=40, decel=4000, tmax=20.911, leave=0.5, reach=0.5}
  [875] = {accel=40, decel=4000, tmax=20.778, leave=0.5, reach=0.5}
  [876] = {accel=40, decel=4000, tmax=20.615, leave=0.5, reach=0.5}
  [877] = {accel=40, decel=4000, tmax=20.432, leave=0.5, reach=0.5}
  [878] = {accel=40, decel=4000, tmax=20.241, leave=0.5, reach=0.5}
  [879] = {accel=40, decel=4000, tmax=20.051, leave=0.5, reach=0.5}
  [880] = {accel=40, decel=4000, tmax=19.864, leave=0.5, reach=0.5}
  [881] = {accel=40, decel=4000, tmax=19.674, leave=0.5, reach=0.5}
  [882] = {accel=40, decel=4000, tmax=19.474, leave=0.5, reach=0.5}
  [883] = {accel=40, decel=4000, tmax=19.254, leave=0.5, reach=0.5}
  [884] = {accel=40, decel=4000, tmax=19.008, leave=0.5, reach=0.5}
  [885] = {accel=40, decel=4000, tmax=18.74, leave=0.5, reach=0.5}
  [886] = {accel=40, decel=4000, tmax=18.459, leave=0.5, reach=0.5}
  [887] = {accel=40, decel=4000, tmax=18.177, leave=0.5, reach=0.5}
  [888] = {accel=40, decel=4000, tmax=17.902, leave=0.5, reach=0.5}
  [889] = {accel=40, decel=4000, tmax=17.636, leave=0.5, reach=0.5}
  [890] = {accel=40, decel=4000, tmax=17.372, leave=0.5, reach=0.5}
  [891] = {accel=40, decel=4000, tmax=17.099, leave=0.5, reach=0.5}
  [892] = {accel=40, decel=4000, tmax=16.81, leave=0.5, reach=0.5}
  [893] = {accel=40, decel=4000, tmax=16.498, leave=0.5, reach=0.5}
  [894] = {accel=40, decel=4000, tmax=16.154, leave=0.5, reach=0.5}
  [895] = {accel=40, decel=4000, tmax=15.767, leave=0.5, reach=0.5}
  [896] = {accel=40, decel=4000, tmax=15.333, leave=0.5, reach=0.5}
  [897] = {accel=40, decel=4000, tmax=14.859, leave=0.5, reach=0.5}
  [898] = {accel=40, decel=4000, tmax=14.358, leave=0.5, reach=0.5}
  [899] = {accel=40, decel=4000, tmax=13.845, leave=0.5, reach=0.5}
  [900] = {accel=40, decel=4000, tmax=13.334, leave=0.5, reach=0.5}
  [901] = {accel=40, decel=4000, tmax=12.837, leave=0.5, reach=0.5}
  [902] = {accel=40, decel=4000, tmax=28.463, leave=0.5, reach=0.5}
  [903] = {accel=40, decel=4000, tmax=13.133, leave=0.5, reach=0.5}
  [904] = {accel=40, decel=4000, tmax=13.624, leave=0.5, reach=0.5}
  [905] = {accel=40, decel=4000, tmax=14.118, leave=0.5, reach=0.5}
  [906] = {accel=40, decel=4000, tmax=14.602, leave=0.5, reach=0.5}
  [907] = {accel=40, decel=4000, tmax=15.062, leave=0.5, reach=0.5}
  [908] = {accel=40, decel=4000, tmax=15.487, leave=0.5, reach=0.5}
  [909] = {accel=40, decel=4000, tmax=15.874, leave=0.5, reach=0.5}
  [910] = {accel=40, decel=4000, tmax=16.227, leave=0.5, reach=0.5}
  [911] = {accel=40, decel=4000, tmax=16.551, leave=0.5, reach=0.5}
  [912] = {accel=40, decel=4000, tmax=16.854, leave=0.5, reach=0.5}
  [913] = {accel=40, decel=4000, tmax=17.146, leave=0.5, reach=0.5}
  [914] = {accel=40, decel=4000, tmax=17.439, leave=0.5, reach=0.5}
  [915] = {accel=40, decel=4000, tmax=17.742, leave=0.5, reach=0.5}
  [916] = {accel=40, decel=4000, tmax=18.055, leave=0.5, reach=0.5}
  [917] = {accel=40, decel=4000, tmax=18.37, leave=0.5, reach=0.5}
  [918] = {accel=40, decel=4000, tmax=18.675, leave=0.5, reach=0.5}
  [919] = {accel=40, decel=4000, tmax=18.962, leave=0.5, reach=0.5}
  [920] = {accel=40, decel=4000, tmax=19.23, leave=0.5, reach=0.5}
  [921] = {accel=40, decel=4000, tmax=19.483, leave=0.5, reach=0.5}
  [922] = {accel=40, decel=4000, tmax=19.725, leave=0.5, reach=0.5}
  [923] = {accel=40, decel=4000, tmax=19.961, leave=0.5, reach=0.5}
  [924] = {accel=40, decel=4000, tmax=20.191, leave=0.5, reach=0.5}
  [925] = {accel=40, decel=4000, tmax=20.416, leave=0.5, reach=0.5}
  [926] = {accel=40, decel=4000, tmax=20.629, leave=0.5, reach=0.5}
  [927] = {accel=40, decel=4000, tmax=20.822, leave=0.5, reach=0.5}
  [928] = {accel=40, decel=4000, tmax=20.985, leave=0.5, reach=0.5}
  [929] = {accel=40, decel=4000, tmax=21.119, leave=0.5, reach=0.5}
  [930] = {accel=40, decel=4000, tmax=21.227, leave=0.5, reach=0.5}
  [931] = {accel=40, decel=4000, tmax=21.316, leave=0.5, reach=0.5}
  [932] = {accel=40, decel=4000, tmax=21.389, leave=0.5, reach=0.5}
  [933] = {accel=40, decel=4000, tmax=21.447, leave=0.5, reach=0.5}
  [934] = {accel=40, decel=4000, tmax=21.495, leave=0.5, reach=0.5}
  [935] = {accel=40, decel=4000, tmax=21.537, leave=0, reach=0.5}
  [936] = {accel=40, decel=4000, tmax=21.58, leave=0, reach=0.5}
  [937] = {accel=40, decel=4000, tmax=21.628, leave=0, reach=0.5}
  [938] = {accel=40, decel=4000, tmax=21.678, leave=0, reach=0.5}
  [939] = {accel=40, decel=4000, tmax=21.723, leave=0, reach=0.5}
  [940] = {accel=40, decel=4000, tmax=21.759, leave=0, reach=0.5}
  [941] = {accel=40, decel=4000, tmax=21.787, leave=0, reach=0.5}
  [942] = {accel=40, decel=4000, tmax=21.811, leave=0, reach=0.5}
  [943] = {accel=40, decel=4000, tmax=21.835, leave=0, reach=0.5}
  [944] = {accel=40, decel=4000, tmax=21.856, leave=0, reach=0.5}
  [945] = {accel=40, decel=4000, tmax=21.866, leave=0, reach=0.5}
  [946] = {accel=40, decel=4000, tmax=21.851, leave=0, reach=0.5}
  [947] = {accel=40, decel=4000, tmax=21.811, leave=0, reach=0.5}
  [948] = {accel=40, decel=4000, tmax=21.753, leave=0, reach=0.5}
  [949] = {accel=40, decel=4000, tmax=21.681, leave=0, reach=0.5}
  [950] = {accel=40, decel=4000, tmax=21.587, leave=0, reach=0.5}
  [951] = {accel=40, decel=4000, tmax=21.452, leave=0, reach=0.5}
  [952] = {accel=40, decel=4000, tmax=21.268, leave=0, reach=0.5}
  [953] = {accel=40, decel=4000, tmax=21.04, leave=0, reach=0.5}
  [954] = {accel=40, decel=4000, tmax=20.796, leave=0, reach=0.5}
  [955] = {accel=40, decel=4000, tmax=20.569, leave=0, reach=0.5}
  [956] = {accel=40, decel=4000, tmax=20.387, leave=0, reach=0.5}
  [957] = {accel=40, decel=4000, tmax=20.263, leave=0, reach=0.5}
  [958] = {accel=40, decel=4000, tmax=20.184, leave=0, reach=0.5}
  [959] = {accel=40, decel=4000, tmax=20.128, leave=0, reach=0.5}
  [960] = {accel=40, decel=4000, tmax=20.074, leave=0, reach=0.5}
  [961] = {accel=40, decel=4000, tmax=20.02, leave=0, reach=0.5}
  [962] = {accel=40, decel=4000, tmax=19.981, leave=0, reach=0.5}
  [963] = {accel=40, decel=4000, tmax=19.963, leave=0, reach=0.5}
  [964] = {accel=40, decel=4000, tmax=19.956, leave=0, reach=0.5}
  [965] = {accel=40, decel=4000, tmax=19.944, leave=0, reach=0.5}
  [966] = {accel=40, decel=4000, tmax=19.922, leave=0, reach=0.5}
  [967] = {accel=40, decel=4000, tmax=19.896, leave=0, reach=0.5}
  [968] = {accel=40, decel=4000, tmax=19.876, leave=0, reach=0.5}
  [969] = {accel=40, decel=4000, tmax=19.87, leave=0, reach=0.5}
  [970] = {accel=40, decel=4000, tmax=19.884, leave=0, reach=0.5}
  [971] = {accel=40, decel=4000, tmax=19.919, leave=0, reach=0.5}
  [972] = {accel=40, decel=4000, tmax=19.969, leave=0, reach=0.5}
  [973] = {accel=40, decel=4000, tmax=20.025, leave=0, reach=0.5}
  [974] = {accel=40, decel=4000, tmax=20.082, leave=0, reach=0.5}
  [975] = {accel=40, decel=4000, tmax=20.142, leave=0, reach=0.5}
  [976] = {accel=40, decel=4000, tmax=20.204, leave=0, reach=0.5}
  [977] = {accel=40, decel=4000, tmax=20.265, leave=0, reach=0.5}
  [978] = {accel=40, decel=4000, tmax=20.323, leave=0, reach=0.5}
  [979] = {accel=40, decel=4000, tmax=20.375, leave=0, reach=0.5}
  [980] = {accel=40, decel=4000, tmax=20.423, leave=0, reach=0.5}
  [981] = {accel=40, decel=4000, tmax=20.462, leave=0, reach=0.5}
  [982] = {accel=40, decel=4000, tmax=20.491, leave=0, reach=0.5}
  [983] = {accel=40, decel=4000, tmax=20.507, leave=0, reach=0.5}
  [984] = {accel=40, decel=4000, tmax=20.507, leave=0, reach=0.5}
  [985] = {accel=40, decel=4000, tmax=20.489, leave=0, reach=0.5}
  [986] = {accel=40, decel=4000, tmax=20.442, leave=0, reach=0.5}
  [987] = {accel=40, decel=4000, tmax=20.359, leave=0, reach=0.5}
  [988] = {accel=40, decel=4000, tmax=20.229, leave=0, reach=0.5}
  [989] = {accel=40, decel=4000, tmax=20.047, leave=0, reach=0.5}
  [990] = {accel=40, decel=4000, tmax=19.808, leave=0, reach=0.5}
  [991] = {accel=40, decel=4000, tmax=19.509, leave=0, reach=0.5}
  [992] = {accel=40, decel=4000, tmax=19.141, leave=0, reach=0.5}
  [993] = {accel=40, decel=4000, tmax=18.69, leave=0, reach=0.5}
  [994] = {accel=40, decel=4000, tmax=18.151, leave=0, reach=0.5}
  [995] = {accel=40, decel=4000, tmax=17.531, leave=0, reach=0.5}
  [996] = {accel=40, decel=4000, tmax=16.849, leave=0, reach=0.5}
  [997] = {accel=40, decel=4000, tmax=16.128, leave=0, reach=0.5}
  [998] = {accel=40, decel=4000, tmax=15.378, leave=0, reach=0.5}
  [999] = {accel=40, decel=4000, tmax=33.87, leave=0, reach=0.5}
num K = 35
num nCountCycle = 1
public num nCurrentTraj = 1
num nCurtRadius
num nDistToOrign = 225.000310635
num nFileId
num nFileId2 = 1
num nHundredRead
num nHundredWrite
public num nMoveID = 10874.554884
public num nPrdRadius = 149.632927
num nPtBuffer = 500
num nPtOfTraj[16] = 11833
num nReadJnt = 1
public num nReadPtr = 934
public num nSpdOfTCP = 2.0910834
public num nTabSpdCode
public num nThousandRead = 10
public num nThousandWrite = 11
num nTime[2]
  [0] = 1611.967
  [1] = -4198.782
public num nTotalTrajs = 1
public num nTrajofRead
num nWriteJnt = 2
public num nWritePtr = 833
public num nZshift = -50
pointRx pGrinding = {x=-24.52, y=111.089, z=4.526, rx=4.421, ry=-179.062, rz=-65, fatherId=fPrdFrame[0]}
pointRx pPBuff = {x=1609.294798, y=46.814741, z=58.995545, rx=0.56357, ry=179.576697, rz=17.423888, shoulder=lefty, elbow=epositive, wrist=wpositive, fatherId=world[0]}
pointRx pPointRead[1000]
  [0] = {x=66.035, y=112.572, z=6.029, rx=-175.516, ry=2.674, rz=115, fatherId=fPrdFrame[0]}
  [1] = {x=64.551, y=112.572, z=5.96, rx=-175.516, ry=2.615, rz=115, fatherId=fPrdFrame[0]}
  [2] = {x=63.066, y=112.572, z=5.892, rx=-175.516, ry=2.555, rz=115, fatherId=fPrdFrame[0]}
  [3] = {x=61.582, y=112.572, z=5.826, rx=-175.517, ry=2.496, rz=115, fatherId=fPrdFrame[0]}
  [4] = {x=60.097, y=112.572, z=5.761, rx=-175.517, ry=2.437, rz=115, fatherId=fPrdFrame[0]}
  [5] = {x=58.613, y=112.573, z=5.698, rx=-175.517, ry=2.378, rz=115, fatherId=fPrdFrame[0]}
  [6] = {x=57.128, y=112.573, z=5.637, rx=-175.517, ry=2.318, rz=115, fatherId=fPrdFrame[0]}
  [7] = {x=55.644, y=112.573, z=5.577, rx=-175.517, ry=2.259, rz=115, fatherId=fPrdFrame[0]}
  [8] = {x=54.159, y=112.573, z=5.519, rx=-175.517, ry=2.2, rz=115, fatherId=fPrdFrame[0]}
  [9] = {x=52.675, y=112.573, z=5.462, rx=-175.518, ry=2.141, rz=115, fatherId=fPrdFrame[0]}
  [10] = {x=51.19, y=112.573, z=5.406, rx=-175.518, ry=2.081, rz=115, fatherId=fPrdFrame[0]}
  [11] = {x=49.706, y=112.573, z=5.353, rx=-175.518, ry=2.022, rz=115, fatherId=fPrdFrame[0]}
  [12] = {x=48.221, y=112.573, z=5.3, rx=-175.518, ry=1.963, rz=115, fatherId=fPrdFrame[0]}
  [13] = {x=46.737, y=112.573, z=5.25, rx=-175.518, ry=1.904, rz=115, fatherId=fPrdFrame[0]}
  [14] = {x=45.252, y=112.573, z=5.201, rx=-175.518, ry=1.844, rz=115, fatherId=fPrdFrame[0]}
  [15] = {x=43.768, y=112.573, z=5.153, rx=-175.519, ry=1.785, rz=115, fatherId=fPrdFrame[0]}
  [16] = {x=42.283, y=112.573, z=5.107, rx=-175.519, ry=1.726, rz=115, fatherId=fPrdFrame[0]}
  [17] = {x=40.799, y=112.573, z=5.063, rx=-175.519, ry=1.667, rz=115, fatherId=fPrdFrame[0]}
  [18] = {x=39.314, y=112.573, z=5.02, rx=-175.519, ry=1.608, rz=115, fatherId=fPrdFrame[0]}
  [19] = {x=37.83, y=112.573, z=4.979, rx=-175.519, ry=1.548, rz=115, fatherId=fPrdFrame[0]}
  [20] = {x=36.345, y=112.573, z=4.939, rx=-175.519, ry=1.489, rz=115, fatherId=fPrdFrame[0]}
  [21] = {x=34.861, y=112.573, z=4.901, rx=-175.519, ry=1.43, rz=115, fatherId=fPrdFrame[0]}
  [22] = {x=33.376, y=112.573, z=4.864, rx=-175.519, ry=1.371, rz=115, fatherId=fPrdFrame[0]}
  [23] = {x=31.892, y=112.573, z=4.829, rx=-175.52, ry=1.312, rz=115, fatherId=fPrdFrame[0]}
  [24] = {x=30.407, y=112.573, z=4.795, rx=-175.52, ry=1.252, rz=115, fatherId=fPrdFrame[0]}
  [25] = {x=28.923, y=112.573, z=4.763, rx=-175.52, ry=1.193, rz=115, fatherId=fPrdFrame[0]}
  [26] = {x=27.438, y=112.573, z=4.733, rx=-175.52, ry=1.134, rz=115, fatherId=fPrdFrame[0]}
  [27] = {x=25.954, y=112.573, z=4.704, rx=-175.52, ry=1.075, rz=115, fatherId=fPrdFrame[0]}
  [28] = {x=24.469, y=112.573, z=4.677, rx=-175.52, ry=1.016, rz=115, fatherId=fPrdFrame[0]}
  [29] = {x=22.985, y=112.573, z=4.651, rx=-175.52, ry=0.956, rz=115, fatherId=fPrdFrame[0]}
  [30] = {x=21.5, y=112.573, z=4.626, rx=-175.52, ry=0.897, rz=115, fatherId=fPrdFrame[0]}
  [31] = {x=20.016, y=112.573, z=4.604, rx=-175.52, ry=0.838, rz=115, fatherId=fPrdFrame[0]}
  [32] = {x=18.531, y=112.573, z=4.583, rx=-175.52, ry=0.779, rz=115, fatherId=fPrdFrame[0]}
  [33] = {x=17.047, y=112.573, z=4.563, rx=-175.52, ry=0.72, rz=115, fatherId=fPrdFrame[0]}
  [34] = {x=15.562, y=112.573, z=4.545, rx=-175.52, ry=0.66, rz=115, fatherId=fPrdFrame[0]}
  [35] = {x=14.078, y=112.573, z=4.528, rx=-175.521, ry=0.601, rz=115, fatherId=fPrdFrame[0]}
  [36] = {x=12.593, y=112.573, z=4.513, rx=-175.521, ry=0.542, rz=115, fatherId=fPrdFrame[0]}
  [37] = {x=11.109, y=112.573, z=4.5, rx=-175.521, ry=0.483, rz=115, fatherId=fPrdFrame[0]}
  [38] = {x=9.624, y=112.573, z=4.488, rx=-175.521, ry=0.424, rz=115, fatherId=fPrdFrame[0]}
  [39] = {x=8.14, y=112.574, z=4.478, rx=-175.521, ry=0.364, rz=115, fatherId=fPrdFrame[0]}
  [40] = {x=6.655, y=112.574, z=4.469, rx=-175.521, ry=0.305, rz=115, fatherId=fPrdFrame[0]}
  [41] = {x=5.171, y=112.574, z=4.462, rx=-175.521, ry=0.246, rz=115, fatherId=fPrdFrame[0]}
  [42] = {x=3.686, y=112.574, z=4.456, rx=-175.521, ry=0.187, rz=115, fatherId=fPrdFrame[0]}
  [43] = {x=2.202, y=112.574, z=4.452, rx=-175.521, ry=0.128, rz=115, fatherId=fPrdFrame[0]}
  [44] = {x=0.717, y=112.574, z=4.449, rx=-175.521, ry=0.068, rz=115, fatherId=fPrdFrame[0]}
  [45] = {x=-0.767, y=112.574, z=4.448, rx=-175.521, ry=0.009, rz=115, fatherId=fPrdFrame[0]}
  [46] = {x=-2.252, y=112.574, z=4.449, rx=-175.521, ry=-0.05, rz=115, fatherId=fPrdFrame[0]}
  [47] = {x=-3.736, y=112.574, z=4.451, rx=-175.521, ry=-0.109, rz=115, fatherId=fPrdFrame[0]}
  [48] = {x=-5.221, y=112.574, z=4.455, rx=-175.521, ry=-0.168, rz=115, fatherId=fPrdFrame[0]}
  [49] = {x=-6.705, y=112.574, z=4.46, rx=-175.521, ry=-0.227, rz=115, fatherId=fPrdFrame[0]}
  [50] = {x=-8.19, y=112.574, z=4.467, rx=-175.521, ry=-0.287, rz=115, fatherId=fPrdFrame[0]}
  [51] = {x=-9.674, y=112.574, z=4.475, rx=-175.521, ry=-0.346, rz=115, fatherId=fPrdFrame[0]}
  [52] = {x=-11.159, y=112.574, z=4.485, rx=-175.521, ry=-0.405, rz=115, fatherId=fPrdFrame[0]}
  [53] = {x=-12.643, y=112.573, z=4.496, rx=-175.521, ry=-0.464, rz=115, fatherId=fPrdFrame[0]}
  [54] = {x=-14.128, y=112.573, z=4.509, rx=-175.521, ry=-0.523, rz=115, fatherId=fPrdFrame[0]}
  [55] = {x=-15.612, y=112.573, z=4.523, rx=-175.521, ry=-0.583, rz=115, fatherId=fPrdFrame[0]}
  [56] = {x=-17.097, y=112.573, z=4.54, rx=-175.52, ry=-0.642, rz=115, fatherId=fPrdFrame[0]}
  [57] = {x=-18.581, y=112.573, z=4.557, rx=-175.52, ry=-0.701, rz=115, fatherId=fPrdFrame[0]}
  [58] = {x=-20.066, y=112.573, z=4.576, rx=-175.52, ry=-0.76, rz=115, fatherId=fPrdFrame[0]}
  [59] = {x=-21.55, y=112.573, z=4.597, rx=-175.52, ry=-0.819, rz=115, fatherId=fPrdFrame[0]}
  [60] = {x=-23.035, y=112.573, z=4.619, rx=-175.52, ry=-0.879, rz=115, fatherId=fPrdFrame[0]}
  [61] = {x=-24.519, y=112.573, z=4.643, rx=-175.52, ry=-0.938, rz=115, fatherId=fPrdFrame[0]}
  [62] = {x=-26.004, y=112.573, z=4.668, rx=-175.52, ry=-0.997, rz=115, fatherId=fPrdFrame[0]}
  [63] = {x=-27.489, y=112.573, z=4.695, rx=-175.52, ry=-1.056, rz=115, fatherId=fPrdFrame[0]}
  [64] = {x=-28.973, y=112.573, z=4.724, rx=-175.52, ry=-1.115, rz=115, fatherId=fPrdFrame[0]}
  [65] = {x=-30.458, y=112.573, z=4.754, rx=-175.52, ry=-1.175, rz=115, fatherId=fPrdFrame[0]}
  [66] = {x=-31.942, y=112.573, z=4.785, rx=-175.52, ry=-1.234, rz=115, fatherId=fPrdFrame[0]}
  [67] = {x=-33.427, y=112.573, z=4.818, rx=-175.52, ry=-1.293, rz=115, fatherId=fPrdFrame[0]}
  [68] = {x=-34.911, y=112.573, z=4.853, rx=-175.52, ry=-1.352, rz=115, fatherId=fPrdFrame[0]}
  [69] = {x=-36.396, y=112.573, z=4.889, rx=-175.519, ry=-1.411, rz=115, fatherId=fPrdFrame[0]}
  [70] = {x=-37.88, y=112.573, z=4.927, rx=-175.519, ry=-1.471, rz=115, fatherId=fPrdFrame[0]}
  [71] = {x=-39.365, y=112.573, z=4.966, rx=-175.519, ry=-1.53, rz=115, fatherId=fPrdFrame[0]}
  [72] = {x=-40.849, y=112.573, z=5.007, rx=-175.519, ry=-1.589, rz=115, fatherId=fPrdFrame[0]}
  [73] = {x=-42.334, y=112.573, z=5.049, rx=-175.519, ry=-1.648, rz=115, fatherId=fPrdFrame[0]}
  [74] = {x=-43.818, y=112.573, z=5.093, rx=-175.519, ry=-1.707, rz=115, fatherId=fPrdFrame[0]}
  [75] = {x=-45.303, y=112.573, z=5.139, rx=-175.519, ry=-1.767, rz=115, fatherId=fPrdFrame[0]}
  [76] = {x=-46.787, y=112.573, z=5.186, rx=-175.518, ry=-1.826, rz=115, fatherId=fPrdFrame[0]}
  [77] = {x=-48.272, y=112.573, z=5.234, rx=-175.518, ry=-1.885, rz=115, fatherId=fPrdFrame[0]}
  [78] = {x=-49.756, y=112.573, z=5.284, rx=-175.518, ry=-1.944, rz=115, fatherId=fPrdFrame[0]}
  [79] = {x=-51.241, y=112.573, z=5.336, rx=-175.518, ry=-2.004, rz=115, fatherId=fPrdFrame[0]}
  [80] = {x=-52.725, y=112.573, z=5.389, rx=-175.518, ry=-2.063, rz=115, fatherId=fPrdFrame[0]}
  [81] = {x=-54.21, y=112.573, z=5.444, rx=-175.518, ry=-2.122, rz=115, fatherId=fPrdFrame[0]}
  [82] = {x=-55.694, y=112.573, z=5.501, rx=-175.518, ry=-2.181, rz=115, fatherId=fPrdFrame[0]}
  [83] = {x=-57.179, y=112.573, z=5.558, rx=-175.517, ry=-2.241, rz=115, fatherId=fPrdFrame[0]}
  [84] = {x=-58.663, y=112.573, z=5.618, rx=-175.517, ry=-2.3, rz=115, fatherId=fPrdFrame[0]}
  [85] = {x=-60.148, y=112.573, z=5.679, rx=-175.517, ry=-2.359, rz=115, fatherId=fPrdFrame[0]}
  [86] = {x=-61.632, y=112.572, z=5.741, rx=-175.517, ry=-2.418, rz=115, fatherId=fPrdFrame[0]}
  [87] = {x=-63.117, y=112.572, z=5.806, rx=-175.517, ry=-2.477, rz=115, fatherId=fPrdFrame[0]}
  [88] = {x=-64.601, y=112.572, z=5.871, rx=-175.516, ry=-2.537, rz=115, fatherId=fPrdFrame[0]}
  [89] = {x=-66.086, y=112.572, z=5.939, rx=-175.516, ry=-2.596, rz=115, fatherId=fPrdFrame[0]}
  [90] = {x=-67.57, y=112.572, z=6.007, rx=-175.516, ry=-2.655, rz=115, fatherId=fPrdFrame[0]}
  [91] = {x=-69.055, y=112.572, z=6.078, rx=-175.516, ry=-2.714, rz=115, fatherId=fPrdFrame[0]}
  [92] = {x=-70.539, y=112.572, z=6.15, rx=-175.516, ry=-2.774, rz=115, fatherId=fPrdFrame[0]}
  [93] = {x=-67.57, y=114.057, z=6.126, rx=-175.457, ry=-2.655, rz=115, fatherId=fPrdFrame[0]}
  [94] = {x=-66.086, y=114.057, z=6.057, rx=-175.457, ry=-2.596, rz=115, fatherId=fPrdFrame[0]}
  [95] = {x=-64.601, y=114.057, z=5.99, rx=-175.457, ry=-2.537, rz=115, fatherId=fPrdFrame[0]}
  [96] = {x=-63.117, y=114.057, z=5.924, rx=-175.457, ry=-2.478, rz=115, fatherId=fPrdFrame[0]}
  [97] = {x=-61.632, y=114.057, z=5.86, rx=-175.458, ry=-2.418, rz=115, fatherId=fPrdFrame[0]}
  [98] = {x=-60.148, y=114.057, z=5.797, rx=-175.458, ry=-2.359, rz=115, fatherId=fPrdFrame[0]}
  [99] = {x=-58.663, y=114.057, z=5.736, rx=-175.458, ry=-2.3, rz=115, fatherId=fPrdFrame[0]}
  [100] = {x=-57.179, y=114.057, z=5.677, rx=-175.458, ry=-2.241, rz=115, fatherId=fPrdFrame[0]}
  [101] = {x=-55.694, y=114.057, z=5.619, rx=-175.458, ry=-2.181, rz=115, fatherId=fPrdFrame[0]}
  [102] = {x=-54.21, y=114.057, z=5.563, rx=-175.458, ry=-2.122, rz=115, fatherId=fPrdFrame[0]}
  [103] = {x=-52.725, y=114.057, z=5.508, rx=-175.459, ry=-2.063, rz=115, fatherId=fPrdFrame[0]}
  [104] = {x=-51.241, y=114.057, z=5.454, rx=-175.459, ry=-2.004, rz=115, fatherId=fPrdFrame[0]}
  [105] = {x=-49.756, y=114.057, z=5.403, rx=-175.459, ry=-1.945, rz=115, fatherId=fPrdFrame[0]}
  [106] = {x=-48.272, y=114.057, z=5.353, rx=-175.459, ry=-1.885, rz=115, fatherId=fPrdFrame[0]}
  [107] = {x=-46.787, y=114.057, z=5.304, rx=-175.459, ry=-1.826, rz=115, fatherId=fPrdFrame[0]}
  [108] = {x=-45.303, y=114.058, z=5.257, rx=-175.459, ry=-1.767, rz=115, fatherId=fPrdFrame[0]}
  [109] = {x=-43.818, y=114.058, z=5.211, rx=-175.46, ry=-1.708, rz=115, fatherId=fPrdFrame[0]}
  [110] = {x=-42.334, y=114.058, z=5.168, rx=-175.46, ry=-1.648, rz=115, fatherId=fPrdFrame[0]}
  [111] = {x=-40.849, y=114.058, z=5.125, rx=-175.46, ry=-1.589, rz=115, fatherId=fPrdFrame[0]}
  [112] = {x=-39.365, y=114.058, z=5.084, rx=-175.46, ry=-1.53, rz=115, fatherId=fPrdFrame[0]}
  [113] = {x=-37.88, y=114.058, z=5.045, rx=-175.46, ry=-1.471, rz=115, fatherId=fPrdFrame[0]}
  [114] = {x=-36.395, y=114.058, z=5.007, rx=-175.46, ry=-1.412, rz=115, fatherId=fPrdFrame[0]}
  [115] = {x=-34.911, y=114.058, z=4.971, rx=-175.46, ry=-1.352, rz=115, fatherId=fPrdFrame[0]}
  [116] = {x=-33.426, y=114.058, z=4.936, rx=-175.46, ry=-1.293, rz=115, fatherId=fPrdFrame[0]}
  [117] = {x=-31.942, y=114.058, z=4.903, rx=-175.461, ry=-1.234, rz=115, fatherId=fPrdFrame[0]}
  [118] = {x=-30.457, y=114.058, z=4.872, rx=-175.461, ry=-1.175, rz=115, fatherId=fPrdFrame[0]}
  [119] = {x=-28.973, y=114.058, z=4.842, rx=-175.461, ry=-1.116, rz=115, fatherId=fPrdFrame[0]}
  [120] = {x=-27.488, y=114.058, z=4.813, rx=-175.461, ry=-1.056, rz=115, fatherId=fPrdFrame[0]}
  [121] = {x=-26.004, y=114.058, z=4.787, rx=-175.461, ry=-0.997, rz=115, fatherId=fPrdFrame[0]}
  [122] = {x=-24.519, y=114.058, z=4.761, rx=-175.461, ry=-0.938, rz=115, fatherId=fPrdFrame[0]}
  [123] = {x=-23.035, y=114.058, z=4.737, rx=-175.461, ry=-0.879, rz=115, fatherId=fPrdFrame[0]}
  [124] = {x=-21.55, y=114.058, z=4.715, rx=-175.461, ry=-0.819, rz=115, fatherId=fPrdFrame[0]}
  [125] = {x=-20.066, y=114.058, z=4.695, rx=-175.461, ry=-0.76, rz=115, fatherId=fPrdFrame[0]}
  [126] = {x=-18.581, y=114.058, z=4.675, rx=-175.461, ry=-0.701, rz=115, fatherId=fPrdFrame[0]}
  [127] = {x=-17.097, y=114.058, z=4.658, rx=-175.461, ry=-0.642, rz=115, fatherId=fPrdFrame[0]}
  [128] = {x=-15.612, y=114.058, z=4.642, rx=-175.461, ry=-0.583, rz=115, fatherId=fPrdFrame[0]}
  [129] = {x=-14.128, y=114.058, z=4.627, rx=-175.461, ry=-0.523, rz=115, fatherId=fPrdFrame[0]}
  [130] = {x=-12.643, y=114.058, z=4.614, rx=-175.461, ry=-0.464, rz=115, fatherId=fPrdFrame[0]}
  [131] = {x=-11.159, y=114.058, z=4.603, rx=-175.461, ry=-0.405, rz=115, fatherId=fPrdFrame[0]}
  [132] = {x=-9.674, y=114.058, z=4.593, rx=-175.461, ry=-0.346, rz=115, fatherId=fPrdFrame[0]}
  [133] = {x=-8.19, y=114.058, z=4.585, rx=-175.462, ry=-0.287, rz=115, fatherId=fPrdFrame[0]}
  [134] = {x=-6.705, y=114.058, z=4.578, rx=-175.462, ry=-0.228, rz=115, fatherId=fPrdFrame[0]}
  [135] = {x=-5.221, y=114.058, z=4.573, rx=-175.462, ry=-0.168, rz=115, fatherId=fPrdFrame[0]}
  [136] = {x=-3.736, y=114.058, z=4.569, rx=-175.462, ry=-0.109, rz=115, fatherId=fPrdFrame[0]}
  [137] = {x=-2.252, y=114.058, z=4.567, rx=-175.462, ry=-0.05, rz=115, fatherId=fPrdFrame[0]}
  [138] = {x=-0.767, y=114.058, z=4.567, rx=-175.462, ry=0.009, rz=115, fatherId=fPrdFrame[0]}
  [139] = {x=0.717, y=114.058, z=4.568, rx=-175.462, ry=0.068, rz=115, fatherId=fPrdFrame[0]}
  [140] = {x=2.202, y=114.058, z=4.57, rx=-175.462, ry=0.128, rz=115, fatherId=fPrdFrame[0]}
  [141] = {x=3.686, y=114.058, z=4.574, rx=-175.462, ry=0.187, rz=115, fatherId=fPrdFrame[0]}
  [142] = {x=5.171, y=114.058, z=4.58, rx=-175.462, ry=0.246, rz=115, fatherId=fPrdFrame[0]}
  [143] = {x=6.655, y=114.058, z=4.587, rx=-175.461, ry=0.305, rz=115, fatherId=fPrdFrame[0]}
  [144] = {x=8.14, y=114.058, z=4.596, rx=-175.461, ry=0.364, rz=115, fatherId=fPrdFrame[0]}
  [145] = {x=9.624, y=114.058, z=4.606, rx=-175.461, ry=0.424, rz=115, fatherId=fPrdFrame[0]}
  [146] = {x=11.109, y=114.058, z=4.618, rx=-175.461, ry=0.483, rz=115, fatherId=fPrdFrame[0]}
  [147] = {x=12.593, y=114.058, z=4.632, rx=-175.461, ry=0.542, rz=115, fatherId=fPrdFrame[0]}
  [148] = {x=14.078, y=114.058, z=4.647, rx=-175.461, ry=0.601, rz=115, fatherId=fPrdFrame[0]}
  [149] = {x=15.562, y=114.058, z=4.663, rx=-175.461, ry=0.66, rz=115, fatherId=fPrdFrame[0]}
  [150] = {x=17.047, y=114.058, z=4.681, rx=-175.461, ry=0.72, rz=115, fatherId=fPrdFrame[0]}
  [151] = {x=18.531, y=114.058, z=4.701, rx=-175.461, ry=0.779, rz=115, fatherId=fPrdFrame[0]}
  [152] = {x=20.016, y=114.058, z=4.722, rx=-175.461, ry=0.838, rz=115, fatherId=fPrdFrame[0]}
  [153] = {x=21.5, y=114.058, z=4.745, rx=-175.461, ry=0.897, rz=115, fatherId=fPrdFrame[0]}
  [154] = {x=22.985, y=114.058, z=4.769, rx=-175.461, ry=0.956, rz=115, fatherId=fPrdFrame[0]}
  [155] = {x=24.469, y=114.058, z=4.795, rx=-175.461, ry=1.016, rz=115, fatherId=fPrdFrame[0]}
  [156] = {x=25.954, y=114.058, z=4.822, rx=-175.461, ry=1.075, rz=115, fatherId=fPrdFrame[0]}
  [157] = {x=27.438, y=114.058, z=4.851, rx=-175.461, ry=1.134, rz=115, fatherId=fPrdFrame[0]}
  [158] = {x=28.923, y=114.058, z=4.882, rx=-175.461, ry=1.193, rz=115, fatherId=fPrdFrame[0]}
  [159] = {x=30.407, y=114.058, z=4.914, rx=-175.46, ry=1.252, rz=115, fatherId=fPrdFrame[0]}
  [160] = {x=31.892, y=114.058, z=4.947, rx=-175.46, ry=1.312, rz=115, fatherId=fPrdFrame[0]}
  [161] = {x=33.376, y=114.058, z=4.982, rx=-175.46, ry=1.371, rz=115, fatherId=fPrdFrame[0]}
  [162] = {x=34.861, y=114.058, z=5.019, rx=-175.46, ry=1.43, rz=115, fatherId=fPrdFrame[0]}
  [163] = {x=36.345, y=114.058, z=5.057, rx=-175.46, ry=1.489, rz=115, fatherId=fPrdFrame[0]}
  [164] = {x=37.83, y=114.058, z=5.097, rx=-175.46, ry=1.549, rz=115, fatherId=fPrdFrame[0]}
  [165] = {x=39.314, y=114.058, z=5.138, rx=-175.46, ry=1.608, rz=115, fatherId=fPrdFrame[0]}
  [166] = {x=40.799, y=114.058, z=5.181, rx=-175.46, ry=1.667, rz=115, fatherId=fPrdFrame[0]}
  [167] = {x=42.283, y=114.058, z=5.226, rx=-175.46, ry=1.726, rz=115, fatherId=fPrdFrame[0]}
  [168] = {x=43.768, y=114.058, z=5.272, rx=-175.459, ry=1.785, rz=115, fatherId=fPrdFrame[0]}
  [169] = {x=45.252, y=114.057, z=5.319, rx=-175.459, ry=1.845, rz=115, fatherId=fPrdFrame[0]}
  [170] = {x=46.737, y=114.057, z=5.368, rx=-175.459, ry=1.904, rz=115, fatherId=fPrdFrame[0]}
  [171] = {x=48.221, y=114.057, z=5.419, rx=-175.459, ry=1.963, rz=115, fatherId=fPrdFrame[0]}
  [172] = {x=49.706, y=114.057, z=5.471, rx=-175.459, ry=2.022, rz=115, fatherId=fPrdFrame[0]}
  [173] = {x=51.19, y=114.057, z=5.525, rx=-175.459, ry=2.082, rz=115, fatherId=fPrdFrame[0]}
  [174] = {x=52.675, y=114.057, z=5.58, rx=-175.458, ry=2.141, rz=115, fatherId=fPrdFrame[0]}
  [175] = {x=54.159, y=114.057, z=5.637, rx=-175.458, ry=2.2, rz=115, fatherId=fPrdFrame[0]}
  [176] = {x=55.644, y=114.057, z=5.695, rx=-175.458, ry=2.259, rz=115, fatherId=fPrdFrame[0]}
  [177] = {x=57.128, y=114.057, z=5.755, rx=-175.458, ry=2.319, rz=115, fatherId=fPrdFrame[0]}
  [178] = {x=58.613, y=114.057, z=5.817, rx=-175.458, ry=2.378, rz=115, fatherId=fPrdFrame[0]}
  [179] = {x=60.097, y=114.057, z=5.88, rx=-175.457, ry=2.437, rz=115, fatherId=fPrdFrame[0]}
  [180] = {x=61.582, y=114.057, z=5.944, rx=-175.457, ry=2.496, rz=115, fatherId=fPrdFrame[0]}
  [181] = {x=63.066, y=114.057, z=6.011, rx=-175.457, ry=2.556, rz=115, fatherId=fPrdFrame[0]}
  [182] = {x=64.551, y=114.057, z=6.078, rx=-175.457, ry=2.615, rz=115, fatherId=fPrdFrame[0]}
  [183] = {x=61.582, y=115.541, z=6.064, rx=-175.398, ry=2.496, rz=115, fatherId=fPrdFrame[0]}
  [184] = {x=60.097, y=115.542, z=6, rx=-175.398, ry=2.437, rz=115, fatherId=fPrdFrame[0]}
  [185] = {x=58.613, y=115.542, z=5.937, rx=-175.398, ry=2.378, rz=115, fatherId=fPrdFrame[0]}
  [186] = {x=57.128, y=115.542, z=5.875, rx=-175.399, ry=2.319, rz=115, fatherId=fPrdFrame[0]}
  [187] = {x=55.644, y=115.542, z=5.815, rx=-175.399, ry=2.259, rz=115, fatherId=fPrdFrame[0]}
  [188] = {x=54.159, y=115.542, z=5.757, rx=-175.399, ry=2.2, rz=115, fatherId=fPrdFrame[0]}
  [189] = {x=52.675, y=115.542, z=5.7, rx=-175.399, ry=2.141, rz=115, fatherId=fPrdFrame[0]}
  [190] = {x=51.19, y=115.542, z=5.645, rx=-175.399, ry=2.082, rz=115, fatherId=fPrdFrame[0]}
  [191] = {x=49.706, y=115.542, z=5.591, rx=-175.4, ry=2.022, rz=115, fatherId=fPrdFrame[0]}
  [192] = {x=48.221, y=115.542, z=5.539, rx=-175.4, ry=1.963, rz=115, fatherId=fPrdFrame[0]}
  [193] = {x=46.737, y=115.542, z=5.488, rx=-175.4, ry=1.904, rz=115, fatherId=fPrdFrame[0]}
  [194] = {x=45.252, y=115.542, z=5.439, rx=-175.4, ry=1.845, rz=115, fatherId=fPrdFrame[0]}
  [195] = {x=43.768, y=115.542, z=5.391, rx=-175.4, ry=1.786, rz=115, fatherId=fPrdFrame[0]}
  [196] = {x=42.283, y=115.542, z=5.345, rx=-175.4, ry=1.726, rz=115, fatherId=fPrdFrame[0]}
  [197] = {x=40.799, y=115.542, z=5.301, rx=-175.4, ry=1.667, rz=115, fatherId=fPrdFrame[0]}
  [198] = {x=39.314, y=115.542, z=5.258, rx=-175.401, ry=1.608, rz=115, fatherId=fPrdFrame[0]}
  [199] = {x=37.83, y=115.542, z=5.217, rx=-175.401, ry=1.549, rz=115, fatherId=fPrdFrame[0]}
  [200] = {x=36.345, y=115.542, z=5.177, rx=-175.401, ry=1.489, rz=115, fatherId=fPrdFrame[0]}
  [201] = {x=34.861, y=115.542, z=5.139, rx=-175.401, ry=1.43, rz=115, fatherId=fPrdFrame[0]}
  [202] = {x=33.376, y=115.542, z=5.102, rx=-175.401, ry=1.371, rz=115, fatherId=fPrdFrame[0]}
  [203] = {x=31.892, y=115.542, z=5.067, rx=-175.401, ry=1.312, rz=115, fatherId=fPrdFrame[0]}
  [204] = {x=30.407, y=115.542, z=5.033, rx=-175.401, ry=1.253, rz=115, fatherId=fPrdFrame[0]}
  [205] = {x=28.923, y=115.542, z=5.001, rx=-175.401, ry=1.193, rz=115, fatherId=fPrdFrame[0]}
  [206] = {x=27.438, y=115.542, z=4.971, rx=-175.401, ry=1.134, rz=115, fatherId=fPrdFrame[0]}
  [207] = {x=25.954, y=115.542, z=4.942, rx=-175.402, ry=1.075, rz=115, fatherId=fPrdFrame[0]}
  [208] = {x=24.469, y=115.542, z=4.915, rx=-175.402, ry=1.016, rz=115, fatherId=fPrdFrame[0]}
  [209] = {x=22.985, y=115.542, z=4.889, rx=-175.402, ry=0.957, rz=115, fatherId=fPrdFrame[0]}
  [210] = {x=21.5, y=115.542, z=4.865, rx=-175.402, ry=0.897, rz=115, fatherId=fPrdFrame[0]}
  [211] = {x=20.016, y=115.543, z=4.842, rx=-175.402, ry=0.838, rz=115, fatherId=fPrdFrame[0]}
  [212] = {x=18.531, y=115.543, z=4.821, rx=-175.402, ry=0.779, rz=115, fatherId=fPrdFrame[0]}
  [213] = {x=17.047, y=115.543, z=4.801, rx=-175.402, ry=0.72, rz=115, fatherId=fPrdFrame[0]}
  [214] = {x=15.562, y=115.543, z=4.783, rx=-175.402, ry=0.66, rz=115, fatherId=fPrdFrame[0]}
  [215] = {x=14.078, y=115.543, z=4.766, rx=-175.402, ry=0.601, rz=115, fatherId=fPrdFrame[0]}
  [216] = {x=12.593, y=115.543, z=4.752, rx=-175.402, ry=0.542, rz=115, fatherId=fPrdFrame[0]}
  [217] = {x=11.109, y=115.543, z=4.738, rx=-175.402, ry=0.483, rz=115, fatherId=fPrdFrame[0]}
  [218] = {x=9.624, y=115.543, z=4.726, rx=-175.402, ry=0.424, rz=115, fatherId=fPrdFrame[0]}
  [219] = {x=8.14, y=115.543, z=4.716, rx=-175.402, ry=0.364, rz=115, fatherId=fPrdFrame[0]}
  [220] = {x=6.655, y=115.543, z=4.707, rx=-175.402, ry=0.305, rz=115, fatherId=fPrdFrame[0]}
  [221] = {x=5.171, y=115.543, z=4.7, rx=-175.402, ry=0.246, rz=115, fatherId=fPrdFrame[0]}
  [222] = {x=3.686, y=115.543, z=4.694, rx=-175.402, ry=0.187, rz=115, fatherId=fPrdFrame[0]}
  [223] = {x=2.202, y=115.543, z=4.69, rx=-175.402, ry=0.128, rz=115, fatherId=fPrdFrame[0]}
  [224] = {x=0.717, y=115.543, z=4.688, rx=-175.402, ry=0.068, rz=115, fatherId=fPrdFrame[0]}
  [225] = {x=-0.767, y=115.543, z=4.687, rx=-175.402, ry=0.009, rz=115, fatherId=fPrdFrame[0]}
  [226] = {x=-2.252, y=115.543, z=4.687, rx=-175.402, ry=-0.05, rz=115, fatherId=fPrdFrame[0]}
  [227] = {x=-3.736, y=115.543, z=4.689, rx=-175.402, ry=-0.109, rz=115, fatherId=fPrdFrame[0]}
  [228] = {x=-5.221, y=115.543, z=4.693, rx=-175.402, ry=-0.168, rz=115, fatherId=fPrdFrame[0]}
  [229] = {x=-6.705, y=115.543, z=4.698, rx=-175.402, ry=-0.228, rz=115, fatherId=fPrdFrame[0]}
  [230] = {x=-8.19, y=115.543, z=4.705, rx=-175.402, ry=-0.287, rz=115, fatherId=fPrdFrame[0]}
  [231] = {x=-9.674, y=115.543, z=4.713, rx=-175.402, ry=-0.346, rz=115, fatherId=fPrdFrame[0]}
  [232] = {x=-11.159, y=115.543, z=4.723, rx=-175.402, ry=-0.405, rz=115, fatherId=fPrdFrame[0]}
  [233] = {x=-12.643, y=115.543, z=4.734, rx=-175.402, ry=-0.464, rz=115, fatherId=fPrdFrame[0]}
  [234] = {x=-14.128, y=115.543, z=4.747, rx=-175.402, ry=-0.524, rz=115, fatherId=fPrdFrame[0]}
  [235] = {x=-15.612, y=115.543, z=4.762, rx=-175.402, ry=-0.583, rz=115, fatherId=fPrdFrame[0]}
